(* IEC 61131-3 sources: BLM_BACKGROUND/src/PROGRAM_FILES/FB (part 2) *)

          GENERAL_STATE#STATE_END:
              reset_trace(Code:=TRC_COPY_RAM_ROM);
              CURRENT_STATE:=GENERAL_STATE#STATE_INIT;

      END_CASE;
      OutputState:=CURRENT_STATE;
  END_FUNCTION_BLOCK

  (*{
#ifdef ORBITALE
}*)
FUNCTION_BLOCK ResettingXxOrbita

    VAR_EXTERNAL
      Axes                            		:ARRAY[_FIRST_AXIS#FIRST_AXIS.._FIRST_AXIS#FIRST_AXIS+_CONST_VAR_DEF._MAXIS#MAXAXIS-1] OF ax;
      pm                              		: ARRAY[_FIRST_AXIS#FIRST_AXIS.._FIRST_AXIS#FIRST_AXIS+_CONST_VAR_DEF._MAXIS#MAXAXIS-1] OF AxisParameters;
      AxisInLimitationCouple		          :ARRAY[_FIRST_AXIS#FIRST_AXIS .. _FIRST_AXIS#FIRST_AXIS+_CONST_VAR_DEF._MAXIS#MAXAXIS-1] OF BOOL;
      TubeIntestate                         :SINT;
      ThreadIntext          	            :BOOL;
    END_VAR

    VAR_EXTERNAL CONSTANT
      X1                                : INT;    //Cart X
      X6                                :INT;
      PIPE_NO_INTESTATE                  :SINT;
    END_VAR

    VAR
        PosAx : REF_TO TO_PositioningAxis;
         Asse    :INT;
		CURRENT_STATE		:INT:=GENERAL_STATE#STATE_INIT;
		Homing  :Homing ;
    END_VAR

    VAR_OUTPUT
		OutputState					:INT;
	END_VAR

    (*{
    #ifdef DH4010
    }*)
      Asse:=X6;
    (*{
    #else  //Fine DH4010
    }*)
      Asse:=X1;
   (* {
    #endif  //Fine NO DH4010
    }*)
    PosAx := AsPositioningAxisRef(Axes[Asse].PosAx);
    IF PosAx^.actualPosition<pm[Asse].MA_POS_LIMIT_MINUS OR
        PosAx^.actualPosition>pm[Asse].MA_POS_LIMIT_PLUS THEN
      //Nelle orbitali, in caso l^asse X1 sia fuori dai limite software si esegue un index a 0
      TubeIntestate:=PIPE_NO_INTESTATE;
      ThreadIntext:=FALSE;
      Homing (Asse:=Asse, Quota:=0, Modo:=EnumHomingMode#SET_OFFSET_OF_ABSOLUTE_ENCODER_BY_POSITION);
    END_IF;
  END_FUNCTION_BLOCK
(*{
#endif  //Fine ORBITALE
}*)

/////////////////////////////////////////////////////////////////////////////////////////////////////////
//Esegue l^impostazione dei flag che eseguono l^inversione del conteggio e del riferimento degli assi
//Sono da armonizzare le seguenti funzionalità:
//1) inversione direzione programmabile per ciascun asse mediante il parametro M32100 (-1, 0, +1)
//2) senso di curvatura DX<=>SX non in processo
FUNCTION_BLOCK FB_InversioneSensoAsse
    VAR_INPUT
      Asse  :INT;
      Senso	:INT;
    END_VAR
    VAR
      Dret  :DINT;
          //CURRENT_STATE					:INT:=STATE_INIT;
         // FB_DisableAxes						:FB_FB_DisableAxes;
          //RestartActivationAsse	:FB_RestartActivationAsse;
    END_VAR
      VAR_OUTPUT
          OutputState		:INT;
      END_VAR
      ;
     (* CASE CURRENT_STATE OF
          STATE_INIT:
            IF pm[Asse].ma_Asse_Abilitato=TRUE THEN
                  CURRENT_STATE:=STATE_DISABLEASSI_DISABLE;
              ELSE
                  CURRENT_STATE:=STATE_END;
              END_IF;

          STATE_DISABLEASSI_DISABLE:
              IF (FB_DisableAxes.outputState<>STATE_END) THEN
                  FB_DisableAxes(Asse:=Asse, Regolatore:=INACTIVE);
              ELSE
                  FB_DisableAxes(Asse:=Asse, Regolatore:=INACTIVE);
                  CASE pm[Asse].ma_ax_motion_dir OF
                      0:;
                          {#ifdef CURVATURA}
                              CASE Asse OF
                                  //Nessuna forzatura di direzione si gestisce l^eventuale inversione del
                                  //conteggio e del riferimento DX<=>SX solo per le macchine in cui
                                  //l^operazione è possibile
                                  Y1,Q1:
                                      {#ifdef ELECT_ALL}
                                          ConteggioDXSX(Asse);
                                      {#endif}
                                      {#ifdef ELECTM}
                                          ConteggioDXSX(Asse);
                                      {#endif}
                                      {#ifdef FOUR_RUNNER}
                                          ConteggioDXSX(Asse);
                                      {#endif}
                              END_CASE;
                              CURRENT_STATE:=STATE_INVERSIONEASSE_RESTART;
                          {#else}
                              CURRENT_STATE:=STATE_END;
                          {#endif};

                      NO_INVERSIONE:
                          //Flag di inversione a OFF
                          {#ifdef CURVATURA}
                              CASE Asse OF
                                  Y1,Q1{#ifdef MATRICE_ELETTRICA},Y2{#endif}:
                                      IF Senso=CURVATURA_DX THEN
                                          Assi[Asse].PosAx.SetConfigData.TypeOfAxis.numberofencoders.encoder_1.inverscountdirection.encoderFeedbackPolarity:=NO;
                                          Assi[Asse].PosAx.setConfigData.TypeOfAxis.SetPointDriverInfo.InvertSetPoint.invSetPoint:=NO;
                                      ELSE
                                          Assi[Asse].PosAx.SetConfigData.TypeOfAxis.numberofencoders.encoder_1.inverscountdirection.encoderFeedbackPolarity:=YES;
                                          Assi[Asse].PosAx.setConfigData.TypeOfAxis.SetPointDriverInfo.InvertSetPoint.invSetPoint:=YES;
                                      END_IF;
                                  ELSE
                                      Assi[Asse].PosAx.SetConfigData.TypeOfAxis.numberofencoders.encoder_1.inverscountdirection.encoderFeedbackPolarity:=NO;
                                      Assi[Asse].PosAx.setConfigData.TypeOfAxis.SetPointDriverInfo.InvertSetPoint.invSetPoint:=NO;
                                      IF Assi[Asse].PosAx.SetConfigData.TypeOfAxis.numberofencoders.numberofencoders=2 THEN
                                          IF Assi[Asse].PosAx.setconfigdata.TypeOfAxis.NumberOfEncoders.encoder_2.encodermode<>SENSOR_ANALOG THEN
                                              //In caso di secondo encoder vero occorre gestire l^inversione del conteggio che per
                                              //l^EFLEX facciamo diventare il contrario di quello dell^encoder 1.
                                              //DA SISTEMARE CON UNA GESTIONE MIGLIORE SE SARA^ NECESSARIO
                                              Assi[Asse].PosAx.SetConfigData.TypeOfAxis.numberofencoders.encoder_2.inverscountdirection.encoderFeedbackPolarity:=YES;
                                          END_IF;
                                      END_IF;
                              END_CASE;
                              CURRENT_STATE:=STATE_INVERSIONEASSE_RESTART;
                          {#else}	//Fine CURVATURA
                              Assi[Asse].PosAx.SetConfigData.TypeOfAxis.numberofencoders.encoder_1.inverscountdirection.encoderFeedbackPolarity:=NO;
                              Assi[Asse].PosAx.setConfigData.TypeOfAxis.SetPointDriverInfo.InvertSetPoint.invSetPoint:=NO;
                              IF Assi[Asse].PosAx.SetConfigData.TypeOfAxis.numberofencoders.numberofencoders=2 THEN
                                  IF Assi[Asse].PosAx.setconfigdata.TypeOfAxis.NumberOfEncoders.encoder_2.encodermode<>SENSOR_ANALOG THEN
                                      //In caso di secondo encoder vero occorre gestire l^inversione del conteggio che per
                                      //l^EFLEX facciamo diventare il contrario di quello dell^encoder 1.
                                      //DA SISTEMARE CON UNA GESTIONE MIGLIORE SE SARA^ NECESSARIO
                                      Assi[Asse].PosAx.SetConfigData.TypeOfAxis.numberofencoders.encoder_2.inverscountdirection.encoderFeedbackPolarity:=YES;
                                  END_IF;
                              END_IF;
                              CURRENT_STATE:=STATE_INVERSIONEASSE_RESTART;
                          {#endif}	//Fine NO CURVATURA

                      SI_INVERSIONE:;
                          //Flag di inversione a ON
                          {#ifdef CURVATURA}
                              CASE Asse OF
                                  Y1,Q1{#ifdef MATRICE_ELETTRICA},Y2{#endif}:
                                      IF Senso=CURVATURA_DX THEN
                                          Assi[Asse].PosAx.SetConfigData.TypeOfAxis.numberofencoders.encoder_1.inverscountdirection.encoderFeedbackPolarity:=YES;
                                          Assi[Asse].PosAx.setConfigData.TypeOfAxis.SetPointDriverInfo.InvertSetPoint.invSetPoint:=YES;
                                      ELSE
                                          Assi[Asse].PosAx.SetConfigData.TypeOfAxis.numberofencoders.encoder_1.inverscountdirection.encoderFeedbackPolarity:=NO;
                                          Assi[Asse].PosAx.setConfigData.TypeOfAxis.SetPointDriverInfo.InvertSetPoint.invSetPoint:=NO;
                                      END_IF;
                                  ELSE
                                      Assi[Asse].PosAx.SetConfigData.TypeOfAxis.numberofencoders.encoder_1.inverscountdirection.encoderFeedbackPolarity:=YES;
                                      Assi[Asse].PosAx.setConfigData.TypeOfAxis.SetPointDriverInfo.InvertSetPoint.invSetPoint:=YES;
                                      IF Assi[Asse].PosAx.SetConfigData.TypeOfAxis.numberofencoders.numberofencoders=2 THEN
                                          IF Assi[Asse].PosAx.setconfigdata.TypeOfAxis.NumberOfEncoders.encoder_2.encodermode<>SENSOR_ANALOG THEN
                                              //In caso di secondo encoder vero occorre gestire l^inversione del conteggio che per
                                              //l^EFLEX facciamo diventare il contrario di quello dell^encoder 1.
                                              //DA SISTEMARE CON UNA GESTIONE MIGLIORE SE SARA^ NECESSARIO
                                              Assi[Asse].PosAx.SetConfigData.TypeOfAxis.numberofencoders.encoder_2.inverscountdirection.encoderFeedbackPolarity:=NO;
                                          END_IF;
                                      END_IF;
                              END_CASE;
                              CURRENT_STATE:=STATE_INVERSIONEASSE_RESTART;
                          {#else}	//Fine CURVATURA
                              Assi[Asse].PosAx.SetConfigData.TypeOfAxis.numberofencoders.encoder_1.inverscountdirection.encoderFeedbackPolarity:=YES;
                              Assi[Asse].PosAx.setConfigData.TypeOfAxis.SetPointDriverInfo.InvertSetPoint.invSetPoint:=YES;
                              IF Assi[Asse].PosAx.SetConfigData.TypeOfAxis.numberofencoders.numberofencoders=2 THEN
                                  IF Assi[Asse].PosAx.setconfigdata.TypeOfAxis.NumberOfEncoders.encoder_2.encodermode<>SENSOR_ANALOG THEN
                                      //In caso di secondo encoder vero occorre gestire l^inversione del conteggio che per
                                      //l^EFLEX facciamo diventare il contrario di quello dell^encoder 1.
                                      //DA SISTEMARE CON UNA GESTIONE MIGLIORE SE SARA^ NECESSARIO
                                      Assi[Asse].PosAx.SetConfigData.TypeOfAxis.numberofencoders.encoder_2.inverscountdirection.encoderFeedbackPolarity:=NO;
                                  END_IF;
                              END_IF;
                              CURRENT_STATE:=STATE_INVERSIONEASSE_RESTART;
                          {#endif}	//Fine NO CURVATURA
                  END_CASE;
              END_IF;

          STATE_INVERSIONEASSE_RESTART:
              IF (RestartActivationAsse.outputState<>STATE_END) THEN
                  RestartActivationAsse(NumAsse:=Asse, Attesa:=TRUE);
              ELSE
                  RestartActivationAsse(NumAsse:=Asse, Attesa:=TRUE);
                  CURRENT_STATE:=STATE_END;
              END_IF;

          STATE_END:
              CURRENT_STATE:=STATE_INIT;
      END_CASE;
      OutputState:=CURRENT_STATE;*)
  END_FUNCTION_BLOCK

  FUNCTION_BLOCK FB_ManagementBrake

    VAR_EXTERNAL
        Start_read								: BOOL;
        i_sys_ReadingSinamicsInUse              :BOOL;
    END_VAR

    VAR_EXTERNAL CONSTANT
            driveObjectIdConstant               : UINT;
            hardwareIdConstant                  :WORD;
    END_VAR

    VAR_INPUT
      Asse         :INT;
      Stato        :SINT;
    END_VAR

    VAR
        Address 			:DINT;
        dret    			:DINT;
        //Ritorno 			:Ret_write_par;

        CURRENT_STATE					:INT:=GENERAL_STATE#STATE_INIT;
        FB_DisableAxes				    :FB_DisableAxes;
        ScritturaDatiSinamics	        :_WRITE_PARAMETER_SINGL;
    END_VAR

    VAR_OUTPUT
        OutputState	:INT;
    END_VAR

      CASE CURRENT_STATE OF
        GENERAL_STATE#STATE_INIT:
              IF (FB_DisableAxes.outputState<>GENERAL_STATE#STATE_END) THEN
                  //Occorre disabilitare l^asse altrimenti il nuovo firmware non accetta il comando
                  FB_DisableAxes(Asse:=Asse (*Regolatore:=INACTIVE*));
              ELSE
                  FB_DisableAxes(Asse:=Asse (*Regolatore:=INACTIVE*));
                (*Address:=UDINT_TO_DINT(Assi[Asse].PosAx.setconfigdata.TypeOfAxis.SetPointDriverInfo.logAddressIn);*)
                  CURRENT_STATE:=_FB_ManagementBrake#STATE_MANAGEMENT_BRAKE_WAIT_READING_SYNAMICS;
              END_IF;

        _FB_ManagementBrake#STATE_MANAGEMENT_BRAKE_WAIT_READING_SYNAMICS:
              IF NOT i_sys_ReadingSinamicsInUse THEN
                  CURRENT_STATE:=_FB_ManagementBrake#STATE_MANAGEMENT_BRAKE_WRITE_SYNAMICS;
              END_IF;

        _FB_ManagementBrake#STATE_MANAGEMENT_BRAKE_WRITE_SYNAMICS:

                IF NOT ScritturaDatiSinamics.Done THEN
                    ScritturaDatiSinamics(Start := Start_read,
                                        driveObjectId :=driveObjectIdConstant,
                                        hardwareId := hardwareIdConstant,
                                        parameterNumber:=uint#1215,
                                        index:=uint#0,
                                        value:=Stato);
                ELSIF ScritturaDatiSinamics.Done THEN
                    ScritturaDatiSinamics(Start := Start_read,
                                        driveObjectId :=driveObjectIdConstant,
                                        hardwareId := hardwareIdConstant,
                                        parameterNumber:=uint#1215,
                                        index:=uint#0,
                                        value:=Stato);
                    ScritturaDatiSinamics.Start :=false;
                    CURRENT_STATE:=GENERAL_STATE#STATE_END;
                ELSIF ScritturaDatiSinamics.error THEN
                    ScritturaDatiSinamics.Start :=false;
                END_IF;
      END_CASE;
    //Occorre disabilitare l^asse altrimenti il nuovo firmware non accetta il comando
    FB_DisableAxes(Asse:=Asse (*Regolatore:=INACTIVE*));
    (*Address:=UDINT_TO_DINT(Assi[Asse].PosAx.setconfigdata.TypeOfAxis.SetPointDriverInfo.logAddressIn);*)
    WHILE i_sys_ReadingSinamicsInUse=TRUE DO ;
      (*dret:=_waitTime(T#0ms); *)
    END_WHILE;

    IF NOT ScritturaDatiSinamics.Done THEN
        ScritturaDatiSinamics(Start := Start_read,
                            driveObjectId :=driveObjectIdConstant,
                            hardwareId := hardwareIdConstant,
                            parameterNumber:=uint#1215,
                            index:=uint#0,
                            value:=Stato);
    ELSIF ScritturaDatiSinamics.Done THEN
        ScritturaDatiSinamics.Start :=false;
    ELSIF ScritturaDatiSinamics.error THEN
        ScritturaDatiSinamics.Start :=false;
    END_IF;
  END_FUNCTION_BLOCK
(*{
#ifdef RUNNER
}*)
	FUNCTION_BLOCK Module_2Axes

        VAR_EXTERNAL
            ModeSpecialReturnCuttingOrbital 	:INT;
            Axes                            :ARRAY[_FIRST_AXIS#FIRST_AXIS.._FIRST_AXIS#FIRST_AXIS+_CONST_VAR_DEF._MAXIS#MAXAXIS-1] OF ax;
            pm                              : ARRAY[_FIRST_AXIS#FIRST_AXIS.._FIRST_AXIS#FIRST_AXIS+_CONST_VAR_DEF._MAXIS#MAXAXIS-1] OF AxisParameters;
        END_VAR

        VAR_EXTERNAL CONSTANT
            INACTIVE_DEACTIVATABLE_AXIS             :SINT;
        END_VAR

		VAR_INPUT
			Asse1          :INT;
			Asse2          :INT;
			Attesa         :BOOL;
		END_VAR

		VAR
            ResetMotionResetAxis				:FB_ResetMotionResetAxis;
            Homing          :Homing;
            Axes1          : REF_TO TO_SynchronousAxis;
            Axes2          : REF_TO TO_SynchronousAxis;
            Axes1MasterAxis :REF_TO TO_PositioningAxis;
            Axes2MasterAxis :REF_TO TO_PositioningAxis;
			Quota1         :LREAL;
			Quota2         :LREAL;
			QuotaIntera1   :DINT;
			QuotaIntera2   :DINT;
			QuotaIntera    :DINT;
			dret           :DINT;
			Counter        :INT;

			CURRENT_STATE		:INT:=GENERAL_STATE#STATE_INIT;
            ReadPosSlave : ReadPosSlave;
		END_VAR
		VAR_OUTPUT
			OutputState			:INT;
		END_VAR
		CASE CURRENT_STATE OF
			GENERAL_STATE#STATE_INIT:
				IF ModeSpecialReturnCuttingOrbital >0 THEN
                    Axes1:= AsSynchronousAxisRef(Axes[Asse1].PosAx);
                    Axes2:= AsSynchronousAxisRef(Axes[Asse2].PosAx);
                    IF ABS(Axes1^.ActualVelocity )<0.1 AND  ABS(Axes2^. ActualVelocity )<0.1 THEN
					//IF ABS(Axes[Asse1].PosAx.motionStateData.commandVelocity)<0.1 AND  ABS(Assi[Asse2].PosAx.motionStateData.commandVelocity)<0.1 THEN
						CURRENT_STATE:=GENERAL_STATE#STATE_END;
					END_IF;
				ELSE
					IF pm[Asse1].ma_Asse_Abilitato=TRUE AND pm[Asse1].ma_Asse_Installato<>INACTIVE_DEACTIVATABLE_AXIS AND
						 pm[Asse2].ma_Asse_Abilitato=TRUE AND pm[Asse2].ma_Asse_Installato<>INACTIVE_DEACTIVATABLE_AXIS THEN
						 //La funzione viene eseguita solo se i due assi sono abilitati e non disattivati
						 IF Attesa THEN
							//Prima di eseguire il modulo si attende che i due assi raggiungano la posizione prevista dalla camma
                            Axes1MasterAxis:= AsPositioningAxisRef(Axes[Asse1].masteraxis);
							ReadPosSlave(NomeMaster:=Axes[Asse1].masteraxis,
																	 Asse:=Asse1,
																	 PosMaster:=Axes1MasterAxis^.actualposition,
																	 Modo:=_EnumCamPositionMode#ACTUAL,
                                                                     PosSlave=>Quota1);
                            Axes2MasterAxis:= AsPositioningAxisRef(Axes[Asse2].masteraxis);
							ReadPosSlave(NomeMaster:=Axes[Asse2].mastername,
																	 Asse:=Asse2,
																	 PosMaster:=Axes2MasterAxis^.actualposition,
																	 Modo:=_EnumCamPositionMode#ACTUAL,
                                                                     PosSlave=>Quota2);
							Counter:=0;
							CURRENT_STATE:=_Module_2Axes#STATE_MODULE_2AXIS_LOOP_WAITING;
						 ELSE
						 	CURRENT_STATE:=_Module_2Axes#STATE_MODULE_2AXIS_HOMING;
						 END_IF;
					ELSE
						CURRENT_STATE:=GENERAL_STATE#STATE_END;
					END_IF;
				END_IF;

            _Module_2Axes#STATE_MODULE_2AXIS_LOOP_WAITING:
                    Axes1:= AsSynchronousAxisRef(Axes[Asse1].PosAx);
                    Axes2:= AsSynchronousAxisRef(Axes[Asse2].PosAx);
				IF ABS(Axes1^.actualposition-Quota1)>0.001 OR
				   ABS(Axes2^.actualposition-Quota2)>0.001 THEN
					IF counter>50 THEN
						CURRENT_STATE:=_Module_2Axes#STATE_MODULE_2AXIS_RESET_AXIS1;
					(*ELSE
						dret:=_waitTime(T#10ms);	//%%%%
						Counter:=Counter+1;*)
					END_IF;
				ELSE
					CURRENT_STATE:=_Module_2Axes#STATE_MODULE_2AXIS_HOMING;
				END_IF;

            _Module_2Axes#STATE_MODULE_2AXIS_RESET_AXIS1:
				IF (ResetMotionResetAxis.outputState<>GENERAL_STATE#STATE_END) THEN
					ResetMotionResetAxis(Asse:=Asse1);
				ELSE
					ResetMotionResetAxis(Asse:=Asse1);
					CURRENT_STATE:=_Module_2Axes#STATE_MODULE_2AXIS_RESET_AXIS2;
				END_IF;

            _Module_2Axes#STATE_MODULE_2AXIS_RESET_AXIS2:
				IF (ResetMotionResetAxis.outputState<>GENERAL_STATE#STATE_END) THEN
					ResetMotionResetAxis(Asse:=Asse2);
				ELSE
					ResetMotionResetAxis(Asse:=Asse2);
					CURRENT_STATE:=_Module_2Axes#STATE_MODULE_2AXIS_HOMING;
				END_IF;

            _Module_2Axes#STATE_MODULE_2AXIS_HOMING:
                Axes1:= AsSynchronousAxisRef(Axes[Asse1].PosAx);
                Axes2:= AsSynchronousAxisRef(Axes[Asse2].PosAx);
				//Legge la quota dell^asse direttamente dal sensore di posizione
                Quota1:=Axes1^.StatusSensor[1].position;
				//Quota1:=Axes[Asse1].PosAx.sensordata[1].position;
				QuotaIntera1:=TO_DINT(Quota1/360);
                Quota2:=Axes2^.StatusSensor[1].position;
				//Quota2:=Axes[Asse2].PosAx.sensordata[1].position;
				QuotaIntera2:=TO_DINT(Quota2/360);
				IF ABS(QuotaIntera1)>ABS(QuotaIntera2) THEN
					Quota1:=Quota1-(QuotaIntera1*360);
					Quota2:=quota2-(QuotaIntera1*360);
				ELSE
					Quota1:=Quota1-(QuotaIntera2*360);
					Quota2:=quota2-(QuotaIntera2*360);
				END_IF;
				Homing(Asse:=Asse1, Quota:=Quota1, Modo:=EnumHomingMode#DIRECT_HOMING_ABSOLUTE);
				CURRENT_STATE:=_Module_2Axes#STATE_MODULE_2AXIS_WAITING_HOMING_AXIS1;

            _Module_2Axes#STATE_MODULE_2AXIS_WAITING_HOMING_AXIS1:
                Axes1:= AsSynchronousAxisRef(Axes[Asse1].PosAx);
				IF Axes1^.StatusWord.%X5 THEN
					Homing(Asse:=Asse2, Quota:=Quota2, Modo:=EnumHomingMode#DIRECT_HOMING_ABSOLUTE);
					CURRENT_STATE:=_Module_2Axes#STATE_MODULE_2AXIS_WAITING_HOMING_AXIS2;
				END_IF;

            _Module_2Axes#STATE_MODULE_2AXIS_WAITING_HOMING_AXIS2:
                Axes2:= AsSynchronousAxisRef(Axes[Asse2].PosAx);
				IF Axes2^.StatusWord.%X5 THEN
					CURRENT_STATE:=GENERAL_STATE#STATE_END;
				END_IF;

			GENERAL_STATE#STATE_END:
				CURRENT_STATE:=GENERAL_STATE#STATE_INIT;
		END_CASE;
		OutputState:=CURRENT_STATE;
	END_FUNCTION_BLOCK
(*{
#endif    //Fine RUNNER
}*)

/************************************************************************************************************
 * SUBJECT TO VERIFICATION OF THE ACTIVATION OF THE POWER SUPPLY, ENABLE ALL MACHINE AXES (DRIVE AND POWER) *
 *                                WITH VERIFICATION OF THE ACTUAL ACTIVATION                                *
 ************************************************************************************************************/
FUNCTION_BLOCK FB_EnableAssi

    VAR_EXTERNAL
        MinuteSavingEnergy                      :INT;
        i_sys_Change_DX_SX                      :BOOL;
        i_sys_enable_Alimen 				    :BOOL;
        i_sys_AutoSetting					    :INT;
        UsoPLCOpen						        :BOOL;
        i_sys_Alimen_Ok 			            :BOOL;
        Axes                                    :ARRAY[_FIRST_AXIS#FIRST_AXIS.._FIRST_AXIS#FIRST_AXIS+_CONST_VAR_DEF._MAXIS#MAXAXIS-1] OF ax;
        pm                                      : ARRAY[_FIRST_AXIS#FIRST_AXIS.._FIRST_AXIS#FIRST_AXIS+_CONST_VAR_DEF._MAXIS#MAXAXIS-1] OF AxisParameters;
        I_VerPLCSafety                          : BYTE;
    END_VAR

    VAR_EXTERNAL CONSTANT
        TRC_MISSING_ADDRESSES_IO            :INT;  //Mancano indirizzi hardware degli I/O
        TRC_MACHINE_DXSX                    :INT;  //Configurazione errata macchina DX SX
        TRC_BASCULANTE_DXSX                   :INT;
        TRC_BASCULANTE_SXDX                   :INT;
        TRC_BASCULANTE_NON_IMPOSTATO          :INT;
        AUTOSETTING_SETTING_SIDE_BASCULANT   :SINT;
        ERR_VERSION_SAFETY                 :DINT;
        VERSIONE_SAFETY                     :BYTE;
        TRC_VIOLATION_BARRIER                 :INT;
        TRC_WAIT_FOR_POWER_SUPPLY_ACTIVATION :INT;
        INACTIVE_DEACTIVATABLE_AXIS         :SINT;
        X1                                  :    INT;    //Cart X
        X2                                  :INT;
        A1                                  :INT;  //Rotation 4RTL/"Rotazione 4RC
        B1                                  :INT;  //Rotation 4RIPC
        INP_PHOTOCELLS_NOT_VIOLATED         :INT;
        TRC_DRIVE                           :INT;  //Azionamento non attivato + numero dellasse
        TRC_POWER                           :INT;  //Potenza non attivata + numero dellasse
        OUT_DRIVES_ON_DPCOUPLER				:INT;
        INP_BARRIER_2                       :INT;
    END_VAR

    VAR_INPUT
      AssiEsclusi		:DWORD:=DWORD#16#FFFFFFFF;
    END_VAR

    VAR
      PosAx  : REF_TO TO_SynchronousAxis;
      masteraxis : REF_TO TO_PositioningAxis;
      i							:INT;
      i2            :INT;
      dret          :DINT;

          CURRENT_STATE									:INT:=GENERAL_STATE#STATE_INIT;
          CURRENT_AXIS									:INT:=-1;
          EnableAxisBLM									:FB_EnableAxisBLM;
          EnableMasterAxisBLM						    :FB_EnableMasterAxisBLM;
          VerificaConfiguraMacchinaDXSX	                :FB_VerificaConfiguraMacchinaDxSx;
    END_VAR
      VAR_OUTPUT
          OutputState	:INT;
          ReturnValue	:BOOL;
      END_VAR
      CASE CURRENT_STATE OF
        GENERAL_STATE#STATE_INIT:
              CURRENT_AXIS:=_FIRST_AXIS#FIRST_AXIS-1;
              StartTimerRisparmioEnergetico(Tempo:=MinuteSavingEnergy);
              CURRENT_STATE:=_FB_EnableAxis#STATE_ENABLEASSI_WAIT_CAMBIO_DX_SX;

        _FB_EnableAxis#STATE_ENABLEASSI_WAIT_CAMBIO_DX_SX:
              IF (i_sys_Change_DX_SX=FALSE) THEN
                  CURRENT_STATE:=_FB_EnableAxis#STATE_ENABLEASSI_WAIT_VERIFICA_IO;
              END_IF;

        _FB_EnableAxis#STATE_ENABLEASSI_WAIT_VERIFICA_IO:
              IF CheckIOAddresses()=TRUE THEN
                  i_sys_enable_alimen:=TRUE;
                  reset_trace(TRC_MISSING_ADDRESSES_IO);
                  (*{#ifdef CURVATURA}*)
                      CURRENT_STATE:=_FB_EnableAxis#STATE_ENABLEASSI_WAIT_VERIFICA_CONFIG_DX_SX;
                  (*{#else}*)
                      CURRENT_STATE:=_FB_EnableAxis#STATE_ENABLEASSI_VERIFICA_SIMULAZIONE;
                  (*{#endif}*)
              ELSE
                  i_sys_enable_alimen:=FALSE;
                  set_trace(Code:=TRC_MISSING_ADDRESSES_IO);
              END_IF;

        _FB_EnableAxis#STATE_ENABLEASSI_WAIT_VERIFICA_CONFIG_DX_SX:
              (*{#ifdef CURVATURA}*)
                  IF (VerificaConfiguraMacchinaDxSx.OutputState<>GENERAL_STATE#STATE_END) THEN
                      VerificaConfiguraMacchinaDxSx();
                  ELSE
                      IF VerificaConfiguraMacchinaDxSx.ReturnValue=TRUE THEN
                          i_sys_enable_alimen:=TRUE;
                          reset_trace(TRC_MACHINE_DXSX);
                          (*{#ifdef SMART}*)
                              CURRENT_STATE:=_FB_EnableAxis#STATE_ENABLEASSI_VERIFICA_BASCULANTE;
                          (*{#else}*)
                              CURRENT_STATE:=_FB_EnableAxis#STATE_ENABLEASSI_VERIFICA_SIMULAZIONE;
                          (*{#endif}*)
                      ELSE
                          i_sys_enable_alimen:=FALSE;
                          set_trace(Code:=TRC_MACHINE_DXSX);
                      END_IF;
                      VerificaConfiguraMacchinaDxSx();
                  END_IF;
              (*{#endif} //FINE CURVATURA*)

        _FB_EnableAxis#STATE_ENABLEASSI_VERIFICA_BASCULANTE:
              (*{#ifdef SMART}*)
                  i:=VerificaBasculanteDxSx();
                  IF i<>2 THEN
                      i_sys_enable_alimen:=FALSE;
                      //VGP destro, configurazione attiva sinistra
                      IF (i=0) THEN
                          IF (i_sys_autosetting<>AUTOSETTING_SETTING_SIDE_BASCULANT) THEN
                              set_trace(Code:=TRC_BASCULANTE_DXSX);
                          END_IF;
                          i2:=i;
                      END_IF;
                      //VGP sinistro, configurazione attiva destra
                      IF (i=1) THEN
                          IF (i_sys_autosetting<>AUTOSETTING_SETTING_SIDE_BASCULANT) THEN
                              set_trace(Code:=TRC_BASCULANTE_SXDX);
                          END_IF;
                          i2:=i;
                      END_IF;
                      //configurazione attiva mancante
                      IF (i=-1) THEN
                          IF (i_sys_autosetting<>AUTOSETTING_SETTING_SIDE_BASCULANT) THEN
                              set_trace(Code:=TRC_BASCULANTE_NON_IMPOSTATO);
                          END_IF;
                          i2:=i;
                      END_IF;
                  ELSE
                      CURRENT_STATE:=_FB_EnableAxis#STATE_ENABLEASSI_VERIFICA_SIMULAZIONE;
                  END_IF;
              (*{#endif}; //FINE SMART*)

        _FB_EnableAxis#STATE_ENABLEASSI_VERIFICA_SIMULAZIONE:
              IF VerificationSimulationAxes()=FALSE THEN
                 (*  {#ifdef PROFINET}
                      {#ifndef EMULAZIONE}*)
                          CURRENT_STATE:=_FB_EnableAxis#STATE_ENABLEASSI_CHECK_VER_SAFETY;
                      (*{#else}	//FINE NO EMULAZIONE*)
                          CURRENT_STATE:=_FB_EnableAxis#STATE_ENABLEASSI_WAIT_BARRIERE_NON_VIOLATE;
                     (*  {#endif} //FINE EMULAZIONE*)
                  (*{#else} //FINE PROFINET*)
                      CURRENT_STATE:=_FB_EnableAxis#STATE_ENABLEASSI_WAIT_BARRIERE_NON_VIOLATE;
                  (*{#endif}; //FINE NO PROFINET*)
              ELSE
                  CURRENT_STATE:=_FB_EnableAxis#STATE_ENABLEASSI_GET_NEXT_STEP;
              END_IF;

        _FB_EnableAxis#STATE_ENABLEASSI_CHECK_VER_SAFETY:
              (*{#ifdef PROFINET}*)
                  IF I_VerPLCSafety<>VERSIONE_SAFETY THEN
                      dret:=Push_Error(code:=ERR_VERSION_SAFETY , Arresto:=TRUE);
                  ELSE
                      CURRENT_STATE:=_FB_EnableAxis#STATE_ENABLEASSI_WAIT_BARRIERE_NON_VIOLATE;
                  END_IF;
              (*{#endif}; //FINE PROFINET*)

        _FB_EnableAxis#STATE_ENABLEASSI_WAIT_BARRIERE_NON_VIOLATE:
              IF (ReadDigitalInput(NumInput:=INP_PHOTOCELLS_NOT_VIOLATED)=TRUE) THEN
                  reset_trace(Code:=TRC_VIOLATION_BARRIER);
                  CURRENT_STATE:=_FB_EnableAxis#STATE_ENABLEASSI_GET_NEXT_STEP;
              ELSE
                  set_trace(Code:=TRC_VIOLATION_BARRIER);
              END_IF;

        _FB_EnableAxis#STATE_ENABLEASSI_GET_NEXT_STEP:
              (*{#ifdef ALIMENTATORE_ACTIVE_LINE}*)
                  CURRENT_STATE:=_FB_EnableAxis#STATE_ENABLEASSI_WAIT_ALIMENTATORE_ON;
              (*{#else}*)
                  CURRENT_STATE:=_FB_EnableAxis#STATE_ENABLEASSI_CHECK_DH4010;
              (*{#endif}*)

        _FB_EnableAxis#STATE_ENABLEASSI_WAIT_ALIMENTATORE_ON:
              (*{#ifdef ALIMENTATORE_ACTIVE_LINE}*)
                  IF (VerificationSimulationAxes()=FALSE AND i_sys_alimen_ok=FALSE) THEN
                      set_trace(Code:=TRC_WAIT_FOR_POWER_SUPPLY_ACTIVATION);
                  ELSE
                      reset_trace(TRC_WAIT_FOR_POWER_SUPPLY_ACTIVATION);
                      CURRENT_STATE:=_FB_EnableAxis#STATE_ENABLEASSI_CHECK_DH4010;
                  END_IF;
              (*{#endif};*)

        _FB_EnableAxis#STATE_ENABLEASSI_CHECK_DH4010:
              (*{#ifdef DH4010}*)
                  CURRENT_STATE:=_FB_EnableAxis#STATE_ENABLEASSI_ENABLE_MASTER_1_DH4010;
              (*{#else}*)
                  CURRENT_STATE:=_FB_EnableAxis#STATE_ENABLEASSI_ENABLE_MASTER;
              (*{#endif};*)

        _FB_EnableAxis#STATE_ENABLEASSI_ENABLE_MASTER_1_DH4010:
              (*{#ifdef DH4010}*)
                masteraxis := AsPositioningAxisRef(Axes[X1].masteraxis);
                IF masteraxis^.StatusWord.%X0 = TRUE THEN
                      IF (USOPLCOpen) THEN
                          IF (EnableMasterAxisBLM.outputState<>GENERAL_STATE#STATE_END) THEN
                              EnableMasterAxisBLM(0(* WHEN_COMMAND_DONE*)); ///Con altri casi e guale
                          ELSE
                              EnableMasterAxisBLM(0 (* , WHEN_COMMAND_DONE*));
                              CURRENT_STATE:=_FB_EnableAxis#STATE_ENABLEASSI_ENABLE_MASTER_2_DH4010;
                          END_IF;
                      ELSE
                          IF (EnableAxisBLM.outputState<>GENERAL_STATE#STATE_END) THEN
                              EnableAxisBlm(Axis:=Axes[X1].masteraxis, NumeroAsse:=-1, (*ModoAttesa:=WHEN_COMMAND_DONE,*) NumMaster:=0);
                          ELSE
                              EnableAxisBlm(Axis:=Axes[X1].masteraxis, NumeroAsse:=-1, (*ModoAttesa:=WHEN_COMMAND_DONE,*) NumMaster:=0);
                              CURRENT_STATE:=_FB_EnableAxis#STATE_ENABLEASSI_ENABLE_MASTER_2_DH4010;
                          END_IF;
                      END_IF;
                  END_IF;
              (*{#endif};*)

        _FB_EnableAxis#STATE_ENABLEASSI_ENABLE_MASTER_2_DH4010:
              (*{#ifdef DH4010}*)
              masteraxis := AsPositioningAxisRef(Axes[X2].masteraxis);
              IF masteraxis^.StatusWord.%X0 = TRUE THEN
                      IF (USOPLCOpen) THEN
                          IF (EnableMasterAxisBLM.outputState<>GENERAL_STATE#STATE_END) THEN
                              EnableMasterAxisBLM(1 (*Axes[X2].masteraxis, WHEN_COMMAND_DONE*));
                          ELSE
                              EnableMasterAxisBLM(1 (*Axes[X2].masteraxis, WHEN_COMMAND_DONE*));
                              CURRENT_STATE:=_FB_EnableAxis#STATE_ENABLEASSI_CHECK_FOUR_RUNNER;
                          END_IF;
                      ELSE
                          IF (EnableAxisBLM.outputState<>GENERAL_STATE#STATE_END) THEN
                              EnableAxisBlm(Axis:=Axes[X2].masteraxis, NumeroAsse:=-1, (*ModoAttesa:=WHEN_COMMAND_DONE,*) NumMaster:=1);
                          ELSE
                              EnableAxisBlm(Axis:=Axes[X2].masteraxis, NumeroAsse:=-1, (*ModoAttesa:=WHEN_COMMAND_DONE,*) NumMaster:=1);
                              CURRENT_STATE:=_FB_EnableAxis#STATE_ENABLEASSI_CHECK_FOUR_RUNNER;
                          END_IF;
                      END_IF;
                  END_IF;
              (*{#endif};*)

        _FB_EnableAxis#STATE_ENABLEASSI_ENABLE_MASTER:
                masteraxis := AsPositioningAxisRef(Axes[X1].masteraxis);
                IF masteraxis^.StatusWord.%X0 = TRUE THEN
                  IF (USOPLCOpen) THEN
                      IF (EnableMasterAxisBLM.outputState<>GENERAL_STATE#STATE_END) THEN
                          EnableMasterAxisBLM(0 (*Axes[X1].masteraxis*));
                      ELSE
                          EnableMasterAxisBLM(0 (* , Axes[X1].masteraxis*));
                          CURRENT_STATE:=_FB_EnableAxis#STATE_ENABLEASSI_CHECK_FOUR_RUNNER;
                      END_IF;
                  ELSE
                      IF (EnableAxisBLM.outputState<>GENERAL_STATE#STATE_END) THEN
                          EnableAxisBlm(Axis:=Axes[X1].masteraxis, NumeroAsse:=-1(* , ModoAttesa:=WHEN_COMMAND_DONE*));
                      ELSE
                          EnableAxisBlm(Axis:=Axes[X1].masteraxis, NumeroAsse:=-1 (* , ModoAttesa:=WHEN_COMMAND_DONE*));
                          CURRENT_STATE:=_FB_EnableAxis#STATE_ENABLEASSI_CHECK_FOUR_RUNNER;
                      END_IF;
                  END_IF;
              ELSE
                  CURRENT_STATE:=_FB_EnableAxis#STATE_ENABLEASSI_CHECK_FOUR_RUNNER;
              END_IF;

        _FB_EnableAxis#STATE_ENABLEASSI_CHECK_FOUR_RUNNER:
              (*{#ifdef FOUR_RUNNER_PLAUNO}
                  {#ifndef PLAUNO_LIGHT}*)
                      CURRENT_STATE:=_FB_EnableAxis#STATE_ENABLEASSI_ENABLE_MASTER_TAGLIO_ESTERNO;
                  (*{#else}*)
                      CURRENT_STATE:=_FB_EnableAxis#STATE_ENABLEASSI_CHECK_RUNNER;
                  (*{#endif}
              {#else}*)
                  CURRENT_STATE:=_FB_EnableAxis#STATE_ENABLEASSI_CHECK_RUNNER;
              (*{#endif};*)

        _FB_EnableAxis#STATE_ENABLEASSI_ENABLE_MASTER_TAGLIO_ESTERNO:
              (*{#ifdef FOUR_RUNNER_PLAUNO}
                  {#ifndef PLAUNO_LIGHT}*)
                        masteraxis := AsPositioningAxisRef(Axes[A1].masteraxis);
                        IF masteraxis^.StatusWord.%X0 = TRUE THEN
                          IF (USOPLCOpen) THEN
                              IF (EnableMasterAxisBLM.outputState<>GENERAL_STATE#STATE_END) THEN
                                  EnableMasterAxisBLM(1 (* , Axes[A1].masteraxis, WHEN_COMMAND_DONE*));
                              ELSE
                                  EnableMasterAxisBLM(1 (* , Axes[A1].masteraxis, WHEN_COMMAND_DONE*));
                                  CURRENT_STATE:=_FB_EnableAxis#STATE_ENABLEASSI_CHECK_RUNNER;
                              END_IF;
                          ELSE
                              IF (EnableAxisBlm.outputState<>GENERAL_STATE#STATE_END) THEN
                                  EnableAxisBlm(Axis:=Axes[A1].masteraxis, NumeroAsse:=-1(* , ModoAttesa:=WHEN_COMMAND_DONE*));
                              ELSE
                                  EnableAxisBlm(Axis:=Axes[A1].masteraxis, NumeroAsse:=-1 (* , ModoAttesa:=WHEN_COMMAND_DONE*));
                                  CURRENT_STATE:=_FB_EnableAxis#STATE_ENABLEASSI_CHECK_RUNNER;
                              END_IF;
                          END_IF;
                      END_IF;
                  (*{#endif};
              {#endif};*)

        _FB_EnableAxis#STATE_ENABLEASSI_CHECK_RUNNER:
              (*{#ifdef RUNNER}
                  {#ifdef B1_B2}*)
                      CURRENT_STATE:=_FB_EnableAxis#STATE_ENABLEASSI_ENABLE_MASTER_TAGLIO_INTERNO;
                  (*{#else}*)
                      CURRENT_STATE:=_FB_EnableAxis#STATE_ENABLEASSI_ENABLE_LOOP;
                  (*{#endif}
              {#else}*)
                  CURRENT_STATE:=_FB_EnableAxis#STATE_ENABLEASSI_ENABLE_LOOP;
              (*{#endif};*)

        _FB_EnableAxis#STATE_ENABLEASSI_ENABLE_MASTER_TAGLIO_INTERNO:
              (*{#ifdef B1_B2}*)
              masteraxis := AsPositioningAxisRef(Axes[B1].masteraxis);
                  IF masteraxis^.StatusWord.%X0 = TRUE THEN
                      IF (USOPLCOpen) THEN
                          IF (EnableMasterAxisBLM.outputState<>GENERAL_STATE#STATE_END) THEN
                              EnableMasterAxisBLM(2 (* , Axes[B1].masteraxis, WHEN_COMMAND_DONE*));
                          ELSE
                              EnableMasterAxisBLM(2(* , Axes[B1].masteraxis, WHEN_COMMAND_DONE*));
                              CURRENT_STATE:=_FB_EnableAxis#STATE_ENABLEASSI_ENABLE_LOOP;
                          END_IF;
                      ELSE
                          IF (EnableAxisBlm.outputState<>GENERAL_STATE#STATE_END) THEN
                              EnableAxisBlm(Axis:=Axes[B1].masteraxis, NumeroAsse:=-1 (* , ModoAttesa:=WHEN_COMMAND_DONE*));
                          ELSE
                              EnableAxisBlm(Axis:=Axes[B1].masteraxis, NumeroAsse:=-1 (* , ModoAttesa:=WHEN_COMMAND_DONE*));
                              CURRENT_STATE:=_FB_EnableAxis#STATE_ENABLEASSI_ENABLE_LOOP;
                          END_IF;
                      END_IF;
                  END_IF;
              (*{#endif};*)

        _FB_EnableAxis#STATE_ENABLEASSI_ENABLE_LOOP:
              CURRENT_AXIS:=CURRENT_AXIS+1;
              IF (CURRENT_AXIS<_MAXIS#MAXAXIS) THEN
                  IF CheckIfTOactive(Axis:=CURRENT_AXIS) THEN
                      IF getBit(AssiEsclusi, TO_USINT(i))=FALSE OR AssiEsclusi=DWORD#16#FFFFFFFF THEN
                        PosAx:=AsSynchronousAxisRef(axes[i].PosAx);//Valore di I
                        IF TestAssePronto(Asse:=i)=FALSE OR
                           PosAx^.StatusWord.%X0 = FALSE OR
                           PosAx^.StatusWord.%X0 = FALSE OR
                           posax^.VirtualAxis.Mode = UDINT#1 THEN
                              CURRENT_STATE:=_FB_EnableAxis#STATE_ENABLEASSI_ENABLE_SINGLE_AXIS;
                          END_IF;
                      END_IF;
                  END_IF;
              ELSE
                  CURRENT_STATE:=_FB_EnableAxis#STATE_ENABLEASSI_RETURNVALUE;
              END_IF;

        _FB_EnableAxis#STATE_ENABLEASSI_ENABLE_SINGLE_AXIS:
              IF (EnableAxisBLM.outputState<>GENERAL_STATE#STATE_END) THEN
                  EnableAxisBlm(Axis:=Axes[CURRENT_AXIS].PosAx, NumeroAsse:=CURRENT_AXIS (* , ModoAttesa:=IMMEDIATELY*));
              ELSE
                  IF (VerificationSimulationAxes()=TRUE) THEN
                      CURRENT_STATE:=_FB_EnableAxis#STATE_ENABLEASSI_ENABLE_SIMULATION_SINGLE_AXIS;
                  ELSE
                      IF pm[i].ma_asse_installato<>INACTIVE_DEACTIVATABLE_AXIS AND pm[i].ma_Asse_Abilitato=TRUE THEN
                          CURRENT_STATE:=_FB_EnableAxis#STATE_ENABLEASSI_WAIT_DRIVESTATE_ACTIVE;
                      ELSE
                          CURRENT_STATE:=_FB_EnableAxis#STATE_ENABLEASSI_ENABLE_LOOP;
                      END_IF;
                  END_IF;
              END_IF;

        _FB_EnableAxis#STATE_ENABLEASSI_ENABLE_SIMULATION_SINGLE_AXIS:
              IF pm[CURRENT_AXIS].ma_asse_installato=INACTIVE_DEACTIVATABLE_AXIS AND pm[CURRENT_AXIS].ma_Asse_Abilitato=TRUE THEN
                 ; //dret:=_enableAxisSimulation(axis:=Axes[CURRENT_AXIS].PosAx,nextCommand:=WHEN_COMMAND_DONE, commandId:=_getCommandId());	//%%%%
              END_IF;
              CURRENT_STATE:=_FB_EnableAxis#STATE_ENABLEASSI_ENABLE_LOOP;

        // _FB_EnableAxis#STATE_ENABLEASSI_WAIT_DRIVESTATE_ACTIVE: %%%%% in attesa
        //       IF Axes[CURRENT_AXIS].PosAx.actormonitoring.drivestate<>INACTIVE THEN
        //           reset_trace(TRC_DRIVE);
        //           IF pm[i].ma_asse_installato<>INACTIVE_DEACTIVATABLE_AXIS THEN
        //               CURRENT_STATE:=_FB_EnableAxis#STATE_ENABLEASSI_WAIT_POWER_ACTIVE;
        //           ELSE
        //               CURRENT_STATE:=_FB_EnableAxis#STATE_ENABLEASSI_WAIT_CONTROL_ACTIVE;
        //           END_IF;
        //       ELSE
        //           set_trace(Code:=TRC_DRIVE, Axis:=CURRENT_AXIS);
        //       END_IF;

        // _FB_EnableAxis#STATE_ENABLEASSI_WAIT_POWER_ACTIVE:
        //       IF Axes[CURRENT_AXIS].PosAx.actormonitoring.power<>INACTIVE THEN

        //           CURRENT_STATE:=_FB_EnableAxis#STATE_ENABLEASSI_WAIT_CONTROL_ACTIVE;
        //       ELSE
        //           set_trace(Code:=TRC_POWER , Axis:=CURRENT_AXIS);
        //       END_IF;

        _FB_EnableAxis#STATE_ENABLEASSI_WAIT_CONTROL_ACTIVE:
              PosAx:=AsSynchronousAxisRef(axes[i].PosAx);//Valore di I
              IF PosAx^.StatusWord.%X0 = FALSE THEN
                  reset_trace(Code:=TRC_POWER );
                  CURRENT_STATE:=_FB_EnableAxis#STATE_ENABLEASSI_ENABLE_LOOP;
              ELSE
                  set_trace(Code:=TRC_POWER , Axis:=CURRENT_AXIS);
              END_IF;

        _FB_EnableAxis#STATE_ENABLEASSI_RETURNVALUE:
              IF VerificationSimulationAxes()=FALSE THEN
                  (*{#ifdef ORBITALE}*)
                      //Verifica che nel frattempo non sia stata violata almeno una delle zone di sicurezza
                      IF readdigitalinput(NumInput:=INP_PHOTOCELLS_NOT_VIOLATED)=TRUE AND readdigitalinput(NumInput:=INP_BARRIER_2)=TRUE THEN
                          ReturnValue:=TRUE;
                      ELSE
                          ReturnValue:=FALSE;
                      END_IF;
                  (*{#else}	//Fine ORBITALE*)
                      //Verifica che nel frattempo non sia stata violata la zona di sicurezza
                      IF readdigitalinput(NumInput:=INP_PHOTOCELLS_NOT_VIOLATED)=TRUE THEN
                          ReturnValue:=TRUE;
                      ELSE
                          ReturnValue:=FALSE;
                      END_IF;
                  (*{#endif} //Fine NO ORBITALE *)
              ELSE
                  ReturnValue:=TRUE;
              END_IF;
              WriteDigitalOutput(NumOutput:=OUT_DRIVES_ON_DPCOUPLER, Value:=ReturnValue);
              CURRENT_STATE:=GENERAL_STATE#STATE_END;

          GENERAL_STATE#STATE_END:
              CURRENT_STATE:=GENERAL_STATE#STATE_INIT;
      END_CASE;
      OutputState:=CURRENT_STATE;
  END_FUNCTION_BLOCK

/*****************************************************************************************
 * VERIFIES THE CORRECT MATCH BETWEEN THE MACHINE'S PROGRAMMING AND THE DX SX STATUS SET *
 *****************************************************************************************/

  FUNCTION_BLOCK FB_VerificaConfiguraMacchinaDxSx

    VAR_EXTERNAL
        Axes                            :ARRAY[_FIRST_AXIS#FIRST_AXIS.._FIRST_AXIS#FIRST_AXIS+_CONST_VAR_DEF._MAXIS#MAXAXIS-1] OF ax;
        pm                              : ARRAY[_FIRST_AXIS#FIRST_AXIS.._FIRST_AXIS#FIRST_AXIS+_CONST_VAR_DEF._MAXIS#MAXAXIS-1] OF AxisParameters;
        i_sys_sense_curve               :INT;		//1=Macchina DX  -1=Macchina SX
    END_VAR

    VAR_EXTERNAL CONSTANT
        Y1 :    INT;  //Y-axis bending arm
        Q1 :    INT;  //Horizontal head
        DX                                              :INT;
    END_VAR

	VAR
		RiferimentoY  :_EnumYesNo;
		EncoderY      :_EnumYesNo;
		RiferimentoQ  :_EnumYesNo;
		EncoderQ      :_EnumYesNo;
		dret          :DINT;
		Esito         :BOOL;

		CURRENT_STATE			:INT:=GENERAL_STATE#STATE_INIT;
		AttesaAvvioSistema:FB_WaitingStartUpSystem;
        AxesY1         :REF_TO TO_SynchronousAxis;
        AxesQ1         :REF_TO TO_SynchronousAxis;
	END_VAR
	VAR_OUTPUT
		OutputState			:INT;
		ReturnValue			:BOOL;
	END_VAR
	(*{#ifdef CURVATURA}*)
		CASE CURRENT_STATE OF
			GENERAL_STATE#STATE_INIT:
				(*{#ifdef DXSX_PROCESSO}*)
					ReturnValue:=TRUE;
					CURRENT_STATE:=GENERAL_STATE#STATE_END;
				(*{#else}*)
					ReturnValue:=FALSE;
					IF (i_sys_sense_curve=0) THEN
						CURRENT_STATE:=GENERAL_STATE#STATE_END;
					ELSE
						CURRENT_STATE:=_FB_VerificaConfiguraMacchinaDxSx#STATE_VERIFICATION_CONFIG_DXSX_WAITING_END_RESTART_Y1;
					END_IF;
				(*{#endif} //FINE NO DXSX_PROCESSO*)

			_FB_VerificaConfiguraMacchinaDxSx#STATE_VERIFICATION_CONFIG_DXSX_WAITING_END_RESTART_Y1:
                AxesY1:= AsSynchronousAxisRef(Axes[Y1].PosAx);
                AxesQ1:= AsSynchronousAxisRef(Axes[Q1].PosAx);
				IF NOT (AxesY1^.StatusWord.%X2  OR AxesQ1^.StatusWord.%X2) THEN
					CURRENT_STATE:=_FB_VerificaConfiguraMacchinaDxSx#STATE_VERIFY_CONFIG_DXSX_WAIT_RESTART_SYSTEM;
				END_IF;

			_FB_VerificaConfiguraMacchinaDxSx#STATE_VERIFY_CONFIG_DXSX_WAIT_RESTART_SYSTEM:
				IF (AttesaAvvioSistema.outputState<>GENERAL_STATE#STATE_END) THEN
					AttesaAvvioSistema(AttesaSimotion:=TRUE, AttesaSinamics:=FALSE);
				ELSE
					AttesaAvvioSistema(AttesaSimotion:=TRUE, AttesaSinamics:=FALSE);

                    AxesY1:= AsSynchronousAxisRef(Axes[Y1].PosAx);
                    IF AxesY1^.Sensor[1].InverseDirection  THEN
                        EncoderY:=_EnumYesNo#YES;
                    ELSE
                        EncoderY:=_EnumYesNo#NO;
                    END_IF;

                    IF AxesY1^.Actor.InverseDirection  THEN
                        RiferimentoY:=_EnumYesNo#YES;
                    ELSE
                        RiferimentoY:=_EnumYesNo#NO;
                    END_IF;

                    AxesQ1:= AsSynchronousAxisRef(Axes[Q1].PosAx);
                    IF AxesQ1^.Sensor[1].InverseDirection  THEN
                        EncoderQ:=_EnumYesNo#YES;
                    ELSE
                        EncoderQ:=_EnumYesNo#NO;
                    END_IF;

                    IF AxesQ1^.Actor.InverseDirection  THEN
                        RiferimentoQ:=_EnumYesNo#YES;
                    ELSE
                        RiferimentoQ:=_EnumYesNo#NO;
                    END_IF;

					//EncoderY:=Axes[Y1].PosAx.ActiveConfigData.TypeOfAxis.NumberOfEncoders.Encoder_1.InversCountDirection.encoderFeedbackPolarity;
					//RiferimentoY:=Axes[Y1].PosAx.ActiveConfigData.TypeOfAxis.SetPointDriverInfo.InvertSetPoint.invSetPoint;
					//EncoderQ:=Axes[Q1].PosAx.ActiveConfigData.TypeOfAxis.NumberOfEncoders.Encoder_1.InversCountDirection.encoderFeedbackPolarity;
					//RiferimentoQ:=Axes[Q1].PosAx.ActiveConfigData.TypeOfAxis.SetPointDriverInfo.InvertSetPoint.invSetPoint;
					CURRENT_STATE:=_FB_VerificaConfiguraMacchinaDxSx#STATE_VERIFY_CONFIG_DXSX_RETURN_VALUE;
				END_IF;

			_FB_VerificaConfiguraMacchinaDxSx#STATE_VERIFY_CONFIG_DXSX_RETURN_VALUE:
				IF i_sys_sense_curve=DX THEN
					//Macchina Destra
					IF pm[Y1].ma_ax_motion_dir>=0 THEN
						//Nessuna inversione Y
						IF EncoderY=_EnumYesNo#NO THEN
							IF RiferimentoY=_EnumYesNo#NO THEN
								IF pm[Q1].ma_ax_motion_dir>=0 THEN
									//Nessuna inversione Q
									IF EncoderQ=_EnumYesNo#NO THEN
										IF RiferimentoQ=_EnumYesNo#NO THEN
											ReturnValue:=TRUE;
										END_IF;
									END_IF;
								ELSE
									//Inversione Q
									IF EncoderQ=_EnumYesNo#YES THEN
										IF RiferimentoQ=_EnumYesNo#YES THEN
											ReturnValue:=TRUE;
										END_IF;
									END_IF;
								END_IF;
							END_IF;
						END_IF;
					ELSE
						//Inversione Y
						IF EncoderY=_EnumYesNo#YES THEN
							IF RiferimentoY=_EnumYesNo#YES THEN
								IF pm[Q1].ma_ax_motion_dir>=0 THEN
									//Nessuna inversione Q
									IF EncoderQ=_EnumYesNo#NO THEN
										IF RiferimentoQ=_EnumYesNo#NO THEN
											ReturnValue:=TRUE;
										END_IF;
									END_IF;
								ELSE
									//Inversione Q
									IF EncoderQ=_EnumYesNo#YES THEN
										IF RiferimentoQ=_EnumYesNo#YES THEN
											ReturnValue:=TRUE;
										END_IF;
									END_IF;
								END_IF;
							END_IF;
						END_IF;
					END_IF;
				ELSE
					//Macchina Sinistra
					IF pm[Y1].ma_ax_motion_dir>=0 THEN
						//Nessuna inversione Y
						IF EncoderY=_EnumYesNo#YES THEN
							IF RiferimentoY=_EnumYesNo#YES THEN
								IF pm[Q1].ma_ax_motion_dir>=0 THEN
									//Nessuna inversione Q
									IF EncoderQ=_EnumYesNo#YES THEN
										IF RiferimentoQ=_EnumYesNo#YES THEN
											ReturnValue:=TRUE;
										END_IF;
									END_IF;
								ELSE
									//Inversione Q
									IF EncoderQ=_EnumYesNo#NO THEN
										IF RiferimentoQ=_EnumYesNo#NO THEN
											ReturnValue:=TRUE;
										END_IF;
									END_IF;
								END_IF;
							END_IF;
						END_IF;
					ELSE
						//Inversione Y
						IF EncoderY=_EnumYesNo#NO THEN
							IF RiferimentoY=_EnumYesNo#NO THEN
								IF pm[Q1].ma_ax_motion_dir>=0 THEN
									//Nessuna inversione Q
									IF EncoderQ=_EnumYesNo#YES THEN
										IF RiferimentoQ=_EnumYesNo#YES THEN
											ReturnValue:=TRUE;
										END_IF;
									END_IF;
								ELSE
									//Inversione Q
									IF EncoderQ=_EnumYesNo#NO THEN
										IF RiferimentoQ=_EnumYesNo#NO THEN
											ReturnValue:=TRUE;
										END_IF;
									END_IF;
								END_IF;
							END_IF;
						END_IF;
					END_IF;
				END_IF;
				CURRENT_STATE:=GENERAL_STATE#STATE_END;

			GENERAL_STATE#STATE_END:
				CURRENT_STATE:=GENERAL_STATE#STATE_INIT;
		END_CASE;
	(*{#else}	//FINE CURVATURA*)
		ReturnValue:=TRUE;
		CURRENT_STATE:=GENERAL_STATE#STATE_END;
	(*{#endif} //FINE NO CURVATURA*)
	OutputState:=CURRENT_STATE;
END_FUNCTION_BLOCK

FUNCTION_BLOCK FB_EnableAxisBlm

    VAR_EXTERNAL
        MinuteSavingEnergy              :INT;
        Axes                            :ARRAY[_FIRST_AXIS#FIRST_AXIS.._FIRST_AXIS#FIRST_AXIS+_CONST_VAR_DEF._MAXIS#MAXAXIS-1] OF ax;
        pm                              : ARRAY[_FIRST_AXIS#FIRST_AXIS.._FIRST_AXIS#FIRST_AXIS+_CONST_VAR_DEF._MAXIS#MAXAXIS-1] OF AxisParameters;
        Start_read						: BOOL;
    END_VAR

    VAR_EXTERNAL CONSTANT
        TRC_WAIT_FOR_POWER_SUPPLY_ACTIVATION    :INT;
        driveObjectIdConstant                   : UINT;
        hardwareIdConstant                      :WORD;
        TRC_DEACTIVATION_SAFETY                 :INT;
        INACTIVE_DEACTIVATABLE_AXIS             :SINT;

    END_VAR

    VAR_INPUT
      Axis        :DB_ANY;
      NumeroAsse  :INT;
      ModoAttesa  :EnumNextCommandEnable;
          NumMaster		:INT:=0;
    END_VAR

    VAR
          simotion_plc    : WORD;
          posax                   : REF_TO TO_SynchronousAxis;
          dret					:DINT;
          Address				:DINT;
          AppoSafety  	:DWORD;
          StatoSafety		:REAL;

          CURRENT_STATE				:INT:=GENERAL_STATE#STATE_INIT;
          EnableSingleAxisBLM	    :FB_EnableSingleAxisBLM;
          DisableAssi			    :FB_DisableAxes;
          LetturaSinamicsREAL       :_READ_PARAMETER_SINGLE;
    END_VAR
      VAR_OUTPUT
          OutputState		:INT;
      END_VAR

      CASE CURRENT_STATE OF
          GENERAL_STATE#STATE_INIT:
              StartTimerRisparmioEnergetico(Tempo:=MinuteSavingEnergy);
              IF NumeroAsse=-1 THEN
                  //Asse Master sempre abilitato
                    posax:= AsSynchronousAxisRef(Axis);
                  IF PosAx^.StatusWord.%X0 = FALSE THEN //enable //.STATUSWORD.%X0
                      CURRENT_STATE:=_FB_EnableSingleAxisBLM#STATE_ENABLESINGLEAXIS_ENABLE;
                  ELSE
                      CURRENT_STATE:=GENERAL_STATE#STATE_END;
                  END_IF;
              ELSE
                posax:= AsSynchronousAxisRef(Axes[NumeroAsse].posax);
                  IF posax^.VirtualAxis.Mode=UDINT#1 THEN
                      CURRENT_STATE:=_FB_EnableSingleAxisBLM#STATE_ENABLESINGLEAXIS_ENABLE;
                  ELSE
                     (*  {#ifdef PROFINET}
                          {#ifndef EMULAZIONE}*)
                              CURRENT_STATE:=_FB_EnableSingleAxisBLM#STATE_ENABLESINGLEAXIS_PROFINET;
                          (*{#else}*)
                              CURRENT_STATE:=_FB_EnableSingleAxisBLM#STATE_ENABLESINGLEAXIS_CHECK_SAFETY_INTEGRATED;
                          (*{#endif}
                      {#else}*)
                          CURRENT_STATE:=_FB_EnableSingleAxisBLM#STATE_ENABLESINGLEAXIS_CHECK_SAFETY_INTEGRATED;
                     (*  {#endif}*)
                  END_IF;
              END_IF;

              _FB_EnableSingleAxisBLM#STATE_ENABLESINGLEAXIS_PROFINET:
              (*{#ifdef PROFINET}*)
                  //Attesa che l^asse non sia in stato safety
                  AppoSafety:=ReadStateSafety(Asse:=NumeroAsse);
                  IF AppoSafety<>DWORD#0 AND pm[NumeroAsse].ma_Asse_Abilitato=TRUE AND ModoAttesa<>EnumNextCommandEnable#IMMEDIATELY THEN
                      CURRENT_STATE:=_FB_EnableSingleAxisBLM#STATE_ENABLESINGLEAXIS_WAIT_EMERGENZA;
                  ELSE
                      CURRENT_STATE:=_FB_EnableSingleAxisBLM#STATE_ENABLESINGLEAXIS_CHECK_SAFETY_INTEGRATED;
                  END_IF;
              (*{#endif};*)

              _FB_EnableSingleAxisBLM#STATE_ENABLESINGLEAXIS_WAIT_EMERGENZA:
             (*  {#ifdef PROFINET}*)
                  AppoSafety:=ReadStateSafety(Asse:=NumeroAsse);
                  IF (getBit(AppoSafety, USINT#5)=TRUE) THEN
                      //In caso di stato di emergenza impostato dal PLC safety
                      //agli azionamenti, occorre indicare all^operatore di premere
                      //e rilasciare il fungo per resettare il PLC safety da
                      //tale condizione
                      set_trace(Code:= TRC_WAIT_FOR_POWER_SUPPLY_ACTIVATION);
                  ELSE
                      Reset_Trace(Code:= TRC_WAIT_FOR_POWER_SUPPLY_ACTIVATION);
                      CURRENT_STATE:=_FB_EnableSingleAxisBLM#STATE_ENABLESINGLEAXIS_WAIT_SAFETY_OFF;
                  END_IF;
              (*{#endif};*)

              _FB_EnableSingleAxisBLM#STATE_ENABLESINGLEAXIS_WAIT_SAFETY_OFF:
              (*{#ifdef PROFINET}*)
                  AppoSafety:=ReadStateSafety(Asse:=NumeroAsse);
                  IF (AppoSafety<>DWORD#0) THEN
                      set_trace(Code:=TRC_DEACTIVATION_SAFETY , Axis:=NumeroAsse);
                  ELSE
                      reset_trace(Code:=TRC_DEACTIVATION_SAFETY );
                      CURRENT_STATE:=_FB_EnableSingleAxisBLM#STATE_ENABLESINGLEAXIS_CHECK_SAFETY_INTEGRATED;
                  END_IF;
              (*{#endif};*)

              _FB_EnableSingleAxisBLM#STATE_ENABLESINGLEAXIS_CHECK_SAFETY_INTEGRATED:
              (*{#ifdef SAFETY_INTEGRATED}*)
                IF VerificationSimulationAxes()=FALSE AND pm[NumeroAsse].ma_asse_installato<>INACTIVE_DEACTIVATABLE_AXIS  THEN
                      //Attende per tutti gli assi attivi che la condizione di safety
                      //venga tolta prima di abilitare l^asse

                     LetturaSinamicsReal(
                                                        driveObjectId := driveObjectIdConstant,
                                                        hardwareId := hardwareIdConstant,
                                                        parameterNumber:=UINT#9722,
                                                        index:=UINT#0,
                                                        Value_REAL=>StatoSafety);
                      CURRENT_STATE:=_FB_EnableSingleAxisBLM#STATE_ENABLESINGLEAXIS_INTEGRATED_WAIT_SAFETY_OFF;
                  ELSE
                      CURRENT_STATE:=_FB_EnableSingleAxisBLM#STATE_ENABLESINGLEAXIS_TESTL1;
                  END_IF;
              (*{#else}*)
                  //CURRENT_STATE:=_FB_EnableSingleAxisBLM#STATE_ENABLESINGLEAXIS_TESTL1;
              (*{#endif};*)

              _FB_EnableSingleAxisBLM#STATE_ENABLESINGLEAXIS_INTEGRATED_WAIT_SAFETY_OFF:
              (*{#ifdef SAFETY_INTEGRATED}*)
                 LetturaSinamicsReal(driveObjectId := driveObjectIdConstant,
                                        hardwareId := hardwareIdConstant,
                                        parameterNumber:=UINT#9722,
                                        index:=UINT#0,
                                        Value_REAL=>StatoSafety);
                  IF getBit(TO_DWORD(StatoSafety),USINT#0)=TRUE OR
                                                          getBit(TO_DWORD(StatoSafety),USINT#1)=TRUE OR
                                                          getBit(TO_DWORD(StatoSafety),USINT#2)=TRUE OR
                                                          getBit(TO_DWORD(StatoSafety),USINT#3)=TRUE THEN
                      set_trace(Code:=TRC_DEACTIVATION_SAFETY , Axis:=NumeroAsse);
                      //Avviso PLC di sicurezza per eventuale ripetizione comando
                      //di reset della safety
                      simotion_plc:=setbit(simotion_plc, USINT#4, TRUE);
                  ELSE
                      simotion_plc:=setbit(simotion_plc, USINT#4, FALSE);
                      reset_trace(Code:=TRC_DEACTIVATION_SAFETY );
                      CURRENT_STATE:=_FB_EnableSingleAxisBLM#STATE_ENABLESINGLEAXIS_TESTL1;
                  END_IF;
              (*{#endif};*)

              _FB_EnableSingleAxisBLM#STATE_ENABLESINGLEAXIS_TESTL1:
        IF NoTestL1(Axis:=NumeroAsse)=TRUE THEN
          //Asse non L1 si abilita anche se è disattivato (sarebbe da migliorare ma occorre un test di verifica)
          IF pm[NumeroAsse].ma_asse_abilitato=TRUE THEN
                      CURRENT_STATE:=_FB_EnableSingleAxisBLM#STATE_ENABLESINGLEAXIS_ENABLE;
          END_IF;
        ELSE
          IF pm[NumeroAsse].ma_asse_installato=INACTIVE_DEACTIVATABLE_AXIS  THEN
            //Asse L1 si disabilita se è disattivato
                      CURRENT_STATE:=_FB_EnableSingleAxisBLM#STATE_ENABLESINGLEAXIS_DISABLE;
          ELSE
            //Asse L1 si abilita solo se non è disattivato
            IF pm[NumeroAsse].ma_asse_abilitato=TRUE THEN
                          CURRENT_STATE:=_FB_EnableSingleAxisBLM#STATE_ENABLESINGLEAXIS_ENABLE;
            END_IF;
          END_IF;
        END_IF;

        _FB_EnableSingleAxisBLM#STATE_ENABLESINGLEAXIS_ENABLE:
              IF (EnableSingleAxisBLM.outputState<>GENERAL_STATE#STATE_END) THEN
                  EnableSingleAxisBLM(NumeroAsse );
                  //EnableSingleAxisBLM(Axis, NumeroAsse (* , ModoAttesa*));
              ELSE
                  EnableSingleAxisBLM(NumeroAsse );
                  //EnableSingleAxisBLM(Axis, NumeroAsse (* , ModoAttesa*));
                  CURRENT_STATE:=GENERAL_STATE#STATE_END;
              END_IF;

        _FB_EnableSingleAxisBLM#STATE_ENABLESINGLEAXIS_DISABLE:
              IF (DisableAssi.outputState<>GENERAL_STATE#STATE_END) THEN
                  DisableAssi(Asse:=NumeroAsse(* , Regolatore:=INACTIVE*));
              ELSE
                  DisableAssi(Asse:=NumeroAsse(* , Regolatore:=INACTIVE*));
                  CURRENT_STATE:=GENERAL_STATE#STATE_END;
              END_IF;

          GENERAL_STATE#STATE_END:
              CURRENT_STATE:=GENERAL_STATE#STATE_INIT;
      END_CASE;
      OutputState:=CURRENT_STATE;
  END_FUNCTION_BLOCK

  FUNCTION_BLOCK FB_SET_Condizione_Move_Asse

    VAR_EXTERNAL
        R_Plus		                            :R_TRIG;
        R_Minus                                 :R_TRIG;
    END_VAR

    VAR_INPUT
      Asse	:INT;
    END_VAR
      VAR
          dret	:DINT;

          SkippedCode			:BOOL:=FALSE;
          CURRENT_STATE		:INT:=GENERAL_STATE#STATE_INIT;
        //   {#ifdef RUNNER} %%%%
        //       Modulo_2Assi		:FB_Modulo_2Assi;
        //   {#endif}
        //   MovimentaPaletta:FB_MovimentaPaletta;
      END_VAR
      VAR_OUTPUT
          OutputState			:INT;
      END_VAR
      CASE CURRENT_STATE OF
          GENERAL_STATE#STATE_INIT:
              IF Asse>=_FIRST_AXIS#FIRST_AXIS AND Asse<=_FIRST_AXIS#FIRST_AXIS+_MAXIS#MAXAXIS-1 THEN
                //   {#ifdef RUNNER} %%%%
                //       {#ifdef ASPO_RUNNER}
                //           IF Asse=X1 AND i_sys_senzatubo=FALSE AND (r_plus.Q=TRUE OR r_minus.Q=TRUE) THEN
                //               //Chiusura rulli trascinamento
                //               Set_Disp(Ndisp:=RULLI_TRASCINAMENTO, Stato:=LAVORO, TimerRisparmio:=TRUE);
                //           END_IF;
                //       {#endif}	//Fine ASPO_RUNNER
                //       {#ifdef FOUR_RUNNER_PLAUNO}
                //           CASE Asse OF
                //               X1,Q1,V1:
                //                   Set_Disp(Ndisp:=FORATURA_MORSA, Stato:=RIPOSO, TimerRisparmio:=FALSE);
                //           END_CASE;
                //           IF Asse=X1 THEN
                //               WriteDigitalOutput(NumOutput:=OUT_ASPO_VERTICALE_NO_ATTREZZAGGIO, Value:=TRUE);
                //               {#ifdef B1_B2}
                //                   IF (Modulo_2Assi.outputState<>STATE_END) THEN
                //                       Modulo_2Assi(Asse1:=B1, Asse2:=B2, Attesa:=FALSE);
                //                       SkippedCode:=TRUE;
                //                       GOTO EsciPrima;
                //                   ELSE
                //                       SkippedCode:=FALSE;
                //                       Modulo_2Assi(Asse1:=B1, Asse2:=B2, Attesa:=FALSE);
                //                   END_IF;
                //               {#endif} //FINE B1_B2
                //           ELSE
                //               WriteDigitalOutput(NumOutput:=OUT_ASPO_VERTICALE_NO_ATTREZZAGGIO, Value:=FALSE);
                //           END_IF;
                //           {#ifndef PLAUNO_LIGHT}
                //               IF TestBloccaggio4RCPresente()=TRUE THEN
                //                   set_disp(Ndisp:=BLOCCAGGIO_4RC, Stato:=RIPOSO, TimerRisparmio:=FALSE);
                //               END_IF;
                //           {#endif}	//FINE NO PLAUNO_LIGHT
                //       {#endif}  //Fine FOUR_RUNNER_PLAUNO
                //       {#ifdef THREE_RUNNER}
                //           IF Asse=X1 THEN
                //               WriteDigitalOutput(NumOutput:=OUT_ASPO_VERTICALE_NO_ATTREZZAGGIO, Value:=TRUE);
                //               {#ifdef B1_B2}
                //                   IF (Modulo_2Assi.outputState<>STATE_END) THEN
                //                       Modulo_2Assi(Asse1:=B1, Asse2:=B2, Attesa:=FALSE);
                //                       SkippedCode:=TRUE;
                //                       GOTO EsciPrima;
                //                   ELSE
                //                       SkippedCode:=FALSE;
                //                       Modulo_2Assi(Asse1:=B1, Asse2:=B2, Attesa:=FALSE);
                //                   END_IF;
                //               {#endif} //FINE B1_B2
                //           ELSE
                //               WriteDigitalOutput(NumOutput:=OUT_ASPO_VERTICALE_NO_ATTREZZAGGIO, Value:=FALSE);
                //           END_IF;
                //       {#endif}  //Fine THREE_RUNNER
                //   {#endif}  //Fine RUNNER
                //   EsciPrima:;
                  IF (SkippedCode=FALSE) THEN
                      IF r_plus.Q=TRUE OR r_minus.Q=TRUE THEN
                          CURRENT_STATE:=_FB_Set_Condizione_Move_Asse#STATE_SET_CONDIZIONE_MOVE_ASSE_PRESSIONE_DIREZIONE;
                    //   ELSE
                    //       {#ifdef DH4010}
                    //           CURRENT_STATE:=STATE_SET_CONDIZIONE_MOVE_ASSE_DH4010_RILASCIO_DIREZIONE;
                    //       {#else}
                    //           CURRENT_STATE:=STATE_END;
                    //        {#endif}
                      END_IF;
                  END_IF;
              ELSE
                  CURRENT_STATE:=GENERAL_STATE#STATE_END;
              END_IF;

        _FB_Set_Condizione_Move_Asse#STATE_SET_CONDIZIONE_MOVE_ASSE_PRESSIONE_DIREZIONE:
            //   CASE Asse OF
                //   {#ifdef ORBITALE}
                    //   {#ifdef EFLEX} %%%%
                    //       X1:
                    //           IF i_sys_SenzaTubo=FALSE THEN
                    //               Set_Disp(Ndisp:=RULLI_TRASCINAMENTO, Stato:=LAVORO, TimerRisparmio:=TRUE);
                    //           END_IF;
                    //   {#endif}  //Fine EFLEX
                    //   {#ifdef DH4010}
                    //       X1,X2,X3,X6:
                    //           IF disp[BLOCCAGGIO_3D].position<>RIPOSO AND disp[BLOCCAGGIO_3D].enable=TRUE THEN
                    //               Set_Disp_Position(Ndisp:=BLOCCAGGIO_3D, Value:=RIPOSO, TimerRisparmio:=TRUE);
                    //           END_IF;
                    //           IF disp[BLOCCAGGIO_2D].position<>RIPOSO AND disp[BLOCCAGGIO_2D].enable=TRUE THEN
                    //               Set_Disp_Position(Ndisp:=BLOCCAGGIO_2D, Value:=RIPOSO, TimerRisparmio:=TRUE);
                    //           END_IF;
                    //           IF disp[PINZA_SX].position<>RIPOSO AND disp[PINZA_SX].enable=TRUE THEN
                    //               Set_Disp_Position(Ndisp:=PINZA_SX, Value:=RIPOSO, TimerRisparmio:=TRUE);
                    //           END_IF;
                    //           IF disp[PINZA_DX].position<>RIPOSO AND disp[PINZA_DX].enable=TRUE THEN
                    //               Set_Disp_Position(Ndisp:=PINZA_DX, Value:=RIPOSO, TimerRisparmio:=TRUE);
                    //           END_IF;
                    //           IF disp[TAGLIO_SX].position<>RIPOSO AND disp[TAGLIO_SX].enable=TRUE THEN
                    //               Set_Disp_Position(Ndisp:=TAGLIO_SX, Value:=RIPOSO, TimerRisparmio:=TRUE);
                    //           END_IF;
                    //           IF disp[TAGLIO_DX].position<>RIPOSO AND disp[TAGLIO_DX].enable=TRUE THEN
                    //               Set_Disp_Position(Ndisp:=TAGLIO_DX, Value:=RIPOSO, TimerRisparmio:=TRUE);
                    //           END_IF;
                    //           IF disp[SMUSSATORE_PINZA].position<>RIPOSO AND disp[SMUSSATORE_PINZA].enable=TRUE THEN
                    //               Set_Disp_Position(Ndisp:=SMUSSATORE_PINZA, Value:=RIPOSO, TimerRisparmio:=TRUE);
                    //           END_IF;
                    //           IF disp[SMUSSATORE_UTENSILE].position<>RIPOSO AND disp[SMUSSATORE_UTENSILE].enable=TRUE THEN
                    //               Set_Disp_Position(Ndisp:=SMUSSATORE_UTENSILE, Value:=RIPOSO, TimerRisparmio:=TRUE);
                    //           END_IF;
                    //           IF Asse=X1 THEN
                    //               GestioneBloccaggioScomparsa(Bloccaggio:=BLOCCAGGIO_SUPPORTO1_SX, Scomparsa:=SCOMPARSA_SUPPORTO1_SX);
                    //               GestioneBloccaggioScomparsa(Bloccaggio:=BLOCCAGGIO_SUPPORTO2_SX, Scomparsa:=SCOMPARSA_SUPPORTO2_SX);
                    //           END_IF;
                    //           IF Asse=X2 OR Asse=X3 THEN
                    //               GestioneBloccaggioScomparsa(Bloccaggio:=BLOCCAGGIO_SUPPORTO1_DX, Scomparsa:=SCOMPARSA_SUPPORTO1_DX);
                    //               GestioneBloccaggioScomparsa(Bloccaggio:=BLOCCAGGIO_SUPPORTO2_DX, Scomparsa:=SCOMPARSA_SUPPORTO2_DX);
                    //           END_IF;
                    //           IF Asse=X6 THEN
                    //               IF TeAspoVersione2()=TRUE THEN
                    //                   WriteDigitalOutput(NumOutput:=OUT_ASPO_VER2_RIPRISTINO_FUNZ_AUTOMATICO, Value:=TRUE);
                    //                   IF ReadDigitalInput(NumInput:=INP_ASPO_VER2_NON_PRONTO, Verifica:=TRUE)=TRUE THEN
                    //                       set_trace(Code:=TRC_ATTESA_ASPO_NON_OK_OFF);
                    //                   ELSE
                    //                       reset_trace(Code:=TRC_ATTESA_ASPO_NON_OK_OFF);
                    //                   END_IF;
                    //                   IF ReadDigitalInput(NumInput:=INP_ASPO_VER2_IN_AUTOMATICO, Verifica:=TRUE)=FALSE AND TestCaricoAspo(Programma:=PROGRAMMA_JOG) THEN
                    //                       set_trace(Code:=TRC_ATTESA_ASPO_IN_MODO_AUTOMATICO);
                    //                   ELSE
                    //                       reset_trace(Code:=TRC_ATTESA_ASPO_IN_MODO_AUTOMATICO);
                    //                   END_IF;
                    //               ELSE
                    //                   reset_trace(Code:=TRC_ATTESA_ASPO_NON_OK_OFF);
                    //                   reset_trace(Code:=TRC_ATTESA_ASPO_IN_MODO_AUTOMATICO);
                    //               END_IF;
                    //               IF i_sys_SenzaTubo=FALSE THEN
                    //                   IF disp[RULLI_TRASCINAMENTO].position<>LAVORO THEN
                    //                       Set_Disp(Ndisp:=RULLI_TRASCINAMENTO, Stato:=LAVORO, TimerRisparmio:=TRUE);
                    //                   END_IF;
                    //               END_IF;
                    //           END_IF;
                    //       Y1,Q1:
                    //           IF Disp[SCOMPARSA_SPALLAMENTO_SX].Position<>RIPOSO THEN
                    //               Set_Disp_Position(Ndisp:=SCOMPARSA_SPALLAMENTO_SX, Value:=RIPOSO, TimerRisparmio:=TRUE);
                    //               CURRENT_STATE:=STATE_SET_CONDIZIONE_MOVE_ASSE_WAIT_TIME_500;
                    //               //dret:=_waitTime(T#500ms);
                    //           END_IF;
                    //       Y2,Q2:
                    //           IF Disp[SCOMPARSA_SPALLAMENTO_DX].Position<>RIPOSO THEN
                    //               Set_Disp_Position(Ndisp:=SCOMPARSA_SPALLAMENTO_DX, Value:=RIPOSO, TimerRisparmio:=TRUE);
                    //               CURRENT_STATE:=STATE_SET_CONDIZIONE_MOVE_ASSE_WAIT_TIME_500;
                    //               //dret:=_waitTime(T#500ms);
                    //           END_IF;
                    //   {#endif}  //Fine DH4010
                    //   {#ifdef FOUR_RUNNER_PLAUNO} %%%%
                    //       X1:
                    //           //Apertura morsa IPC
                    //           Set_Disp(Ndisp:=PINZA_INTERNA, Stato:=RIPOSO, TimerRisparmio:=TRUE);
                    //           RiposoTagliOrbitali(Attesa:=FALSE);
                    //           //Apertura morsa carrello accompagnamento
                    //           Set_Disp_Position(Ndisp:=PINZA_ACCOMPAG_CH_AP, Value:=RIPOSO, TimerRisparmio:=TRUE);
                    //           {#ifdef PLAUNO_PLAUNO_LIGHT}
                    //               Set_Disp_Position(Ndisp:=BLOCCAGGIO_TUBO, Value:=RIPOSO, TimerRisparmio:=TRUE);
                    //           {#endif}  //Fine PLAUNO
                    //   {#endif}  //Fine FOUR_RUNNER_PLAUNO
                    //   {#ifdef TWO_RUNNER}
                    //       X1:
                    //           Set_Disp(Ndisp:=PINZA_CARRO_X1, Stato:=RIPOSO, TimerRisparmio:=TRUE);
                    //   {#endif}  //Fine TWO_RUNNER
                    //   {#ifdef THREE_RUNNER}
                    //       X1:
                    //           Set_Disp(Ndisp:=IPC_MORSA_STRAPPO, Stato:=RIPOSO, TimerRisparmio:=TRUE);
                    //           Set_Disp(Ndisp:=PINZA_INTERNA, Stato:=RIPOSO, TimerRisparmio:=TRUE);
                    //   {#endif}  //Fine THREE_RUNNER
                    //   {#ifdef FOUR_RUNNER}
                    //       Q1, V1:
                    //           IF iaddress[INP_SBLOCCO_DX_SX].Port>-1 AND iaddress[INP_SBLOCCO_DX_SX].Bit>-1 THEN
                    //               Set_Disp(Ndisp:=BLOCCO_CANNOTTO, Stato:=RIPOSO, TimerRisparmio:=TRUE);
                    //           END_IF;
                    //   {#endif} //FINE FOUR_RUNNER
                //   {#else}  //Fine ORBITALE
                //       X1:
                        //   {#ifdef SMART} %%%%
                        //       IF TestBasculanteCarico()=FALSE THEN
                        //           //Basculante non è in posizione di carico si solleva la paletta
                        //           IF (MovimentaPaletta.outputState<>STATE_END) THEN
                        //               MovimentaPaletta(Stato:=LAVORO, Attesa:=FALSE);
                        //           ELSE
                        //               MovimentaPaletta(Stato:=LAVORO, Attesa:=FALSE);
                        //               CURRENT_STATE:=STATE_END;
                        //           END_IF;
                        //       ELSE
                        //           reset_trace(TRC_PALETTA_ALTA);
                        //           CURRENT_STATE:=STATE_END;
                        //       END_IF;
                        //   {#else}  //Fine SMART
                        //       IF (MovimentaPaletta.outputState<>STATE_END) THEN
                        //           MovimentaPaletta(Stato:=LAVORO, Attesa:=FALSE);
                        //       ELSE
                        //           MovimentaPaletta(Stato:=LAVORO, Attesa:=FALSE);
                        //           CURRENT_STATE:=STATE_END;
                        //       END_IF;
                        //   {#endif}  //Fine NO SMART
                //       Z1:
                //           IF (MovimentaPaletta.outputState<>STATE_END) THEN
                //               MovimentaPaletta(Stato:=LAVORO, Attesa:=FALSE);
                //           ELSE
                //               MovimentaPaletta(Stato:=LAVORO, Attesa:=FALSE);
                //               CURRENT_STATE:=STATE_END;
                //           END_IF;
                // //   {#endif}  //Fine NO ORBITALE
            //   ELSE

                CURRENT_STATE:=GENERAL_STATE#STATE_END;
            //   END_CASE;

        _FB_Set_Condizione_Move_Asse#STATE_SET_CONDIZIONE_MOVE_ASSE_WAIT_TIME_500:
              //%%%%%
              CURRENT_STATE:=GENERAL_STATE#STATE_END;

        _FB_Set_Condizione_Move_Asse#STATE_SET_CONDIZIONE_MOVE_ASSE_DH4010_RILASCIO_DIREZIONE:
        //       {#ifdef DH4010} %%%%
        //           IF Asse=X6 AND TeAspoVersione2()=TRUE THEN
        //               IF f_plus.Q=TRUE OR f_minus.Q=TRUE THEN
        //                   //Rilascio + o -
        //                   WriteDigitalOutput(NumOutput:=OUT_ASPO_VER2_RIPRISTINO_FUNZ_AUTOMATICO, Value:=FALSE);
        //                   reset_trace(Code:=TRC_ATTESA_ASPO_NON_OK_OFF);
        //               END_IF;
        //           END_IF;
        //       {#endif};	//Fine DH4010

        //   STATE_END:
              CURRENT_STATE:=GENERAL_STATE#STATE_INIT;

      END_CASE;
      OutputState:=CURRENT_STATE;
  END_FUNCTION_BLOCK

  FUNCTION_BLOCK FB_SET_Condizione_Move_Dispositivo

    VAR_EXTERNAL CONSTANT
        FIRST_DEVICE                          :INT;
    END_VAR

    VAR_INPUT
      Dispositivo :INT;
    END_VAR
    VAR
      dret        :DINT;
      Differenza  :LREAL;

          CURRENT_STATE	:INT:=GENERAL_STATE#STATE_INIT;
        //   PosAxeNoWait	:FB_PosAxeNoWait; %%%%
    END_VAR
      VAR_OUTPUT
          OutputState		:INT;
      END_VAR
      CASE CURRENT_STATE OF
          GENERAL_STATE#STATE_INIT:
              CURRENT_STATE:=GENERAL_STATE#STATE_END;
              IF Dispositivo>=FIRST_DEVICE AND Dispositivo <=FIRST_DEVICE+_MAXDEVICES#MAXDEVICES-1 THEN
            //       {#ifndef EFLEX}
            //           IF i_sys_OPMODE=MDAMODE OR r_plus.Q=TRUE OR r_minus.Q=TRUE THEN
            //               //In caso di override a 0 si evita di chiamare la funzione che esegue lo stacco del filo
            //               //dalla gola della testina in attesa di fine movimento per evitare di superare i tempi
            //               //del background
            //               CASE Dispositivo OF
            //                   {#ifdef DH4010}
            //                       SCOMP_PINZA_SX:
            //                           set_disp_position(Ndisp:=PINZA_SX, Value:=RIPOSO, TimerRisparmio:=TRUE);
            //                       SCOMP_PINZA_DX:
            //                           set_disp_position(Ndisp:=PINZA_DX, Value:=RIPOSO, TimerRisparmio:=TRUE);
            //                       SCOMP_MANIPOLATORE_3D:
            //                           IF disp[BLOCCAGGIO_3D].position<>RIPOSO THEN
            //                               set_disp(Ndisp:=BLOCCAGGIO_3D, Stato:=RIPOSO, TimerRisparmio:=TRUE);
            //                           ELSE
            //                               IF (PosAxeNoWait.outputState<>STATE_END) THEN
            //                                   CURRENT_STATE:=STATE_INIT;
            //                                   PosAxeNoWait(Asse:=Z1, Quota:=65, Accelerazione:=50);
            //                               ELSE
            //                                   PosAxeNoWait(Asse:=Z1, Quota:=65, Accelerazione:=50);
            //                                   CURRENT_STATE:=STATE_END;
            //                               END_IF;
            //                           END_IF;
            //                       SCOMPARSA_SUPPORTO1_SX:
            //                           set_disp(Ndisp:=BLOCCAGGIO_SUPPORTO1_SX, Stato:=RIPOSO, TimerRisparmio:=TRUE);
            //                       SCOMPARSA_SUPPORTO2_SX:
            //                           set_disp(Ndisp:=BLOCCAGGIO_SUPPORTO2_SX, Stato:=RIPOSO, TimerRisparmio:=TRUE);
            //                       SCOMPARSA_SUPPORTO1_DX:
            //                           set_disp(Ndisp:=BLOCCAGGIO_SUPPORTO1_DX, Stato:=RIPOSO, TimerRisparmio:=TRUE);
            //                       SCOMPARSA_SUPPORTO2_DX:
            //                           set_disp(Ndisp:=BLOCCAGGIO_SUPPORTO2_DX, Stato:=RIPOSO, TimerRisparmio:=TRUE);
            //                       SCOMP1_SX, SCOMP2_SX:
            //                           set_disp(Ndisp:=PALPATORE_1_SX, Stato:=RIPOSO, TimerRisparmio:=TRUE);
            //                           set_disp(Ndisp:=PALPATORE_2_SX, Stato:=RIPOSO, TimerRisparmio:=TRUE);
            //                           set_disp(Ndisp:=PALPATORE_3_SX, Stato:=RIPOSO, TimerRisparmio:=TRUE);
            //                           set_disp(Ndisp:=PALPATORE_4_SX, Stato:=RIPOSO, TimerRisparmio:=TRUE);
            //                       SCOMP1_DX, SCOMP2_DX:
            //                           set_disp(Ndisp:=PALPATORE_1_DX, Stato:=RIPOSO, TimerRisparmio:=TRUE);
            //                           set_disp(Ndisp:=PALPATORE_2_DX, Stato:=RIPOSO, TimerRisparmio:=TRUE);
            //                           set_disp(Ndisp:=PALPATORE_3_DX, Stato:=RIPOSO, TimerRisparmio:=TRUE);
            //                           set_disp(Ndisp:=PALPATORE_4_DX, Stato:=RIPOSO, TimerRisparmio:=TRUE);
            //                   {#else}  //Fine DH4010
            //                       {#ifdef RUNNER}
            //                           {#ifdef IPC_DISPOSITIVO}
            //                               IPC_AVANZAMENTO:;
            //                                   IF r_plus.Q=TRUE THEN
            //                                       LubrTaglioIPC(Programma:=PROGRAMMA_JOG, Stato:=TRUE);
            //                                   ELSE
            //                                       IF r_minus.Q=TRUE THEN
            //                                           LubrTaglioIPC(Programma:=PROGRAMMA_JOG, Stato:=FALSE);
            //                                       END_IF;
            //                                   END_IF;
            //                                   set_disp(Ndisp:=IPC_MOTORE, Stato:=LAVORO, TimerRisparmio:=TRUE);
            //                           {#endif}	//Fine IPC_DISPOSITIVO
            //                           {#ifdef A1_A2}
            //                               LEVA_SCARICO:
            //                                   IF TestBloccaggio4RCPresente()=TRUE THEN
            //                                       set_disp(Ndisp:=BLOCCAGGIO_4RC, Stato:=RIPOSO, TimerRisparmio:=FALSE);
            //                                   END_IF;
            //                           {#endif}	//FINE A1_A2
            //                           {#ifdef TWO_RUNNER}
            //                               PINZA_CARRO_X1:;	//Solo per compilare il codice
            //                           {#endif}	//Fine TWO_RUNNER	//Fine TWO_RUNNER
            //                           {#ifdef THREE_RUNNER}
            //                               IPC_STRAPPO:
            //                                   IF r_minus.Q=TRUE THEN
            //                                       set_disp(Ndisp:=IPC_MORSA_STRAPPO, Stato:=RIPOSO, TimerRisparmio:=TRUE);
            //                                   END_IF;
            //                               IPC_STRAPPO_SCARICO:
            //                                   IF r_minus.Q=TRUE THEN
            //                                       set_disp(Ndisp:=IPC_MORSA_STRAPPO, Stato:=RIPOSO, TimerRisparmio:=TRUE);
            //                                       set_disp(Ndisp:=IPC_STRAPPO, Stato:=RIPOSO, TimerRisparmio:=TRUE);
            //                                   END_IF;
            //                           {#endif}  //Fine THREE_RUNNER
            //                       {#else}  //Fine RUNNER
            //                           PALETTA:
            //                               IF Disp[PALETTA].enable THEN
            //                                   IF (PosAxeNoWait.outputState<>STATE_END) THEN
            //                                       PosAxeNoWait(Asse:=Z1, Quota:=0);
            //                                       CURRENT_STATE:=STATE_INIT;
            //                                   ELSE
            //                                       PosAxeNoWait(Asse:=Z1, Quota:=0);
            //                                       CURRENT_STATE:=STATE_END;
            //                                   END_IF;
            //                               END_IF;
            //                           {#ifndef ELECTMRL}
            //                               PINZA_CARICO:
            //                                   IF disp[PINZA_CARICO].enable=TRUE THEN
            //                                       PompatoreCARM7(Stato:=TRUE);
            //                                   END_IF;
            //                           {#endif} //FINE NO ELECTMRL
            //                       {#endif}  //Fine NO RUNNER
            //                   {#endif}  //Fine NO DH4010
            //               END_CASE;
            //           END_IF;
            //       {#endif}  //Fine NO EFLEX;
            //   ELSE
                  CURRENT_STATE:=GENERAL_STATE#STATE_END;
              END_IF;

        GENERAL_STATE#STATE_END:
              CURRENT_STATE:=GENERAL_STATE#STATE_INIT;
      END_CASE;
      OutputState:=CURRENT_STATE;
  END_FUNCTION_BLOCK

/**********************************
 * MANAGES THE JOG OF A REAL AXIS *
 **********************************/
  FUNCTION_BLOCK FB_Jog_Asse

    VAR_EXTERNAL
        Axes                            :ARRAY[_FIRST_AXIS#FIRST_AXIS.._FIRST_AXIS#FIRST_AXIS+_CONST_VAR_DEF._MAXIS#MAXAXIS-1] OF ax;
        pm                              : ARRAY[_FIRST_AXIS#FIRST_AXIS.._FIRST_AXIS#FIRST_AXIS+_CONST_VAR_DEF._MAXIS#MAXAXIS-1] OF AxisParameters;
        mcpi_rapid                      : BOOL;
        i_sys_varinc                    : INT;
        i_sys_monitoring                : INT;
        R_Plus		                    :R_TRIG;
        Clk_Minus	                    :BOOL;
        Clk_Plus                        :BOOL;
        R_Rapid                         :R_TRIG; //fronte salita RAPID
        F_Rapid                         :F_TRIG;
        R_Minus                         :R_TRIG;
        F_Plus                          :F_TRIG;
        F_Minus                         :F_TRIG;
        i_sys_PosFinale				    :ARRAY[(_FIRST_AXIS#FIRST_AXIS) .. (_FIRST_AXIS#FIRST_AXIS+_MAXIS#MAXAXIS -1)] OF LREAL;
        i_sys_ACCESSLEVEL               : INT;
        UsoPLCOpen						:BOOL;
        INC                             :ARRAY[0..5] OF LREAL;
    END_VAR

    VAR_EXTERNAL CONSTANT
        W3                                  :INT;
        ACCESS_MANUTENTORE   	            :SINT;
        TRC_MONITORING_DISABILITATO         :INT;
        TRC_JOG_NON_IN_MONITORING           :INT;  //Macchina non in monitoring o livello di accesso troppo basso
        TRC_SAFETY_JOG_DEVICES       :INT;
        MY_BIG_VALUE_REAL                   :REAL;
        EXTRALIMIT         	                :REAL;
    END_VAR

    VAR_INPUT
      Asse          :INT;
    END_VAR

    VAR
      PosAx         : REF_TO TO_SynchronousAxis;
      jogvel        :LREAL;
      corsa         :LREAL;
      jogacc        :LREAL;
      dret          :DINT;
      pMode         :_EnumPositioningMode;
      AppoDirezione :INT;
      i             :INT;

          CURRENT_STATE				        :INT:=GENERAL_STATE#STATE_INIT;
          CURRENT_AXIS				        :INT;
          ResetMotionResetAxis              :FB_ResetMotionResetAxis;
          PosAsse							:FB_PosAsse;
    END_VAR

      VAR_OUTPUT
          OutputState					:INT;
      END_VAR
      CASE CURRENT_STATE OF
          GENERAL_STATE#STATE_INIT:
              CURRENT_AXIS:=_FIRST_AXIS#FIRST_AXIS-1;
              IF Asse>=_FIRST_AXIS#FIRST_AXIS AND Asse<=_FIRST_AXIS#FIRST_AXIS+_MAXIS#MAXAXIS-1 THEN
                  //Per evitare stop della CPU verifica che Asse contenga un numero valido
                  AzzeramentoDistanceTogo(Asse:=Asse);
                  CURRENT_STATE:=_FB_Jog_Asse#STATE_JOG_ASSE_LOOP_RESET_ASSI;
              ELSE
                  CURRENT_STATE:=GENERAL_STATE#STATE_END;
              END_IF;

            _FB_Jog_Asse#STATE_JOG_ASSE_LOOP_RESET_ASSI:
              CURRENT_AXIS:=CURRENT_AXIS+1;
              IF CURRENT_AXIS<_MAXIS#MAXAXIS THEN
                PosAx:= AsSynchronousAxisRef(Axes[CURRENT_AXIS].PosAx);
                IF PosAx^.StatusPositioning.Distance<>0 AND
                  //IF Axes[CURRENT_AXIS].PosAx.poscommand.distancetogo<>0 AND
          CURRENT_AXIS<>Asse AND posax^.simulation.Mode=UDINT#0 THEN //Axes[CURRENT_AXIS].posax.simulation<>ACTIVE THEN
          ;
            //       {#ifdef SOSTEGNO_ELETTRICO} %%%%
            //           IF CURRENT_AXIS<>S1 THEN
            //   //Serve per azzerare tutti gli assi tranne quello selezionato ed il
            //   //sostegno che si deve poter muovere con X1 e Z1 (tubi non tondi)
            //   CURRENT_STATE:=STATE_JOG_ASSE_RESET_ASSE;
            //           END_IF;
            //       {#else}
            //           CURRENT_STATE:=STATE_JOG_ASSE_RESET_ASSE;
            //       {#endif}
                  END_IF;
              ELSE
                  IF TestVelHoldToRun()=TRUE THEN
                      jogvel:=pm[Asse].ma_Vel_Safety_COMFORT3;
                  ELSE
                      IF mcpi_rapid=FALSE THEN
                          jogvel:=pm[Asse].MA_JOG_VELO*pm[Asse].max_ax_velo/100;
                      ELSE
                          jogvel:=pm[Asse].MA_JOG_VELO_RAPID*pm[Asse].max_ax_velo/100;
                      END_IF;
                  END_IF;
                  jogacc:=pm[Asse].MA_MAX_AX_ACCEL*pm[Asse].MA_JOG_ACC/100;
                //   {#ifdef B1_B2} %%%%
                //       //Gli assi B1 e B2 ache con OVERRIDE 1% sono troppo veloci
                //       IF Asse=B1 OR Asse=B2 THEN
                //           jogvel:=1;
                //       END_IF;
                //   {#endif}  //Fine B1_B2
                //   {#ifdef BLOCCAGGIO_DX}
                //       IF Asse=W3 THEN
                //           AppoDirezione:=SN;
                //       ELSE
                //           AppoDirezione:=SN_SP;
                //       END_IF;
                //   {#else}    //Fine BLOCCAGGIO_DX
                //       AppoDirezione:=SN_SP;
                //   {#endif}    //Fine NO BLOCCAGGIO_DX

                  Axes[Asse].MC_Axes.move_jog_param.Acceleration :=jogacc;
                  Axes[Asse].MC_Axes.move_jog_param.Deceleration :=jogacc;
                  Axes[Asse].MC_Axes.move_jog_param.Velocity :=jogvel;
                  CURRENT_STATE:=_FB_Jog_Asse#STATE_JOG_ASSE_JOG_PURO_POSITIVO;
              END_IF;

        _FB_Jog_Asse#STATE_JOG_ASSE_RESET_ASSE:
              IF (ResetMotionResetAxis.outputState<>GENERAL_STATE#STATE_END) THEN
                  ResetMotionResetAxis(Asse:=CURRENT_AXIS);
              ELSE
                  ResetMotionResetAxis(Asse:=CURRENT_AXIS);
                  CURRENT_STATE:=_FB_Jog_Asse#STATE_JOG_ASSE_LOOP_RESET_ASSI;
              END_IF;

        _FB_Jog_Asse#STATE_JOG_ASSE_JOG_PURO_POSITIVO:
              IF ((r_plus.Q=TRUE) AND (Clk_minus=FALSE)) OR
                   ((Clk_plus=TRUE) AND (Clk_minus=FALSE) AND (f_rapid.Q=TRUE)) OR
                   ((Clk_minus=FALSE) AND (Clk_plus=TRUE) AND (r_rapid.q=TRUE)) THEN
                  IF OK_Condizione_Move_Asse(Asse:=Asse, Direzione:=AppoDirezione) THEN
                      IF i_sys_varinc=0 THEN
                          // è in JOG puro e non incrementale
                          //limite positivo attivo
                          PosAx:= AsSynchronousAxisRef(Axes[asse].PosAx);
                          corsa:=PosAx^.PositionLimits_SW.MaxPosition-EXTRALIMIT;
                          //corsa:=Axes[asse].PosAx.swlimit.plusposition-EXTRALIMIT;
                          pMode:=_EnumPositioningMode#ABSOLUTE;
                      ELSE
                          IF i_sys_varinc>=1 AND i_sys_varinc<=5 THEN
                              // valore fisso
                              corsa := INC[i_sys_varinc];
                              pMode:=_EnumPositioningMode#RELATIVE;
                            //   Axes[Asse].mcJogAxisInfo.Increment:=corsa;
                            //   Axes[Asse].mcJogAxisInfo.ModeInc:=TRUE;
                          ELSE // Quota target
                              // Se la quota supera il fine corsa la limita
                                PosAx:= AsSynchronousAxisRef(Axes[asse].PosAx);
                                IF pm[asse].MA_JOG_TARGET > PosAx^.PositionLimits_SW.MaxPosition  THEN
                                   pm[asse].MA_JOG_TARGET:=PosAx^.PositionLimits_SW.MaxPosition-EXTRALIMIT;
                                END_IF;
                            //   IF pm[asse].MA_JOG_TARGET > Axes[asse].PosAx.swlimit.plusposition THEN
                            //       pm[asse].MA_JOG_TARGET:=Axes[asse].PosAx.swlimit.plusposition-EXTRALIMIT;
                            //   END_IF;
                              // se l^asse è oltre la quota target
                              PosAx:= AsSynchronousAxisRef(Axes[asse].PosAx);
                            //   IF Posax^.actualposition-Axes[Asse].Posax.servosettings.additionalcommandvalue[0]+0.1>pm[asse].MA_JOG_TARGET THEN
                            //       corsa:=PosAx^.PositionLimits_SW.MaxPosition-EXTRALIMIT;
                            //   ELSE
                            //       // valore fisso
                            //       corsa:=pm[asse].MA_JOG_TARGET;
                            //   END_IF;
                              pMode:=_EnumPositioningMode#ABSOLUTE;
                          END_IF;
                      END_IF;
                      IF i_sys_monitoring<>0 OR i_sys_Accesslevel<=ACCESS_MANUTENTORE OR SbloccaMonitoring(Asse:=Asse)=TRUE THEN
                          IF Sbloccamonitoring(Asse:=Asse)=TRUE OR i_sys_monitoring=0 THEN
                              set_trace(Code:=TRC_MONITORING_DISABILITATO);
                          END_IF;
                          //Muove solo se in monitoring o con livello password alto e se l^asse non è oltre il finecorsa positivo
                          PosAx:=AsSynchronousAxisRef(Axes[Asse].Posax);
                          IF Posax^.actualposition+0.01 <  PosAx^.PositionLimits_SW.MaxPosition-EXTRALIMIT THEN //Axes[Asse].PosAx.swlimit.plusposition-EXTRALIMIT THEN
                              TestAsseUtensile(Asse);
                              i_sys_PosFinale[Asse]:=corsa;
                              IF (pMode=_EnumPositioningMode#RELATIVE AND USOPLCOpen) THEN
                                  //Axes[Asse].mcJogAxisInfo.Enable:=TRUE;
                                  Axes[Asse].MC_Axes.move_jog_param.JogForward :=TRUE;
                                  //Axes[Asse].mcJogAxisInfo.Forward:=TRUE;
                              ELSE
                                  CURRENT_STATE:=_FB_Jog_Asse#STATE_JOG_ASSE_POS_ASSE_POSITIVE;
                              END_IF;
                          ELSE
                              CURRENT_STATE:=_FB_Jog_Asse#STATE_JOG_ASSE_JOG_PURO_NEGATIVO;
                          END_IF;
                      ELSE
                          set_trace(Code:=TRC_JOG_NON_IN_MONITORING);
                          CURRENT_STATE:=_FB_Jog_Asse#STATE_JOG_ASSE_JOG_PURO_NEGATIVO;
                      END_IF;
                  END_IF;
              ELSE
                  CURRENT_STATE:=_FB_Jog_Asse#STATE_JOG_ASSE_JOG_PURO_NEGATIVO;
              END_IF;
